KUKA KRL program: EPS_2_25089_SANMH02A_C_20251118074756.src

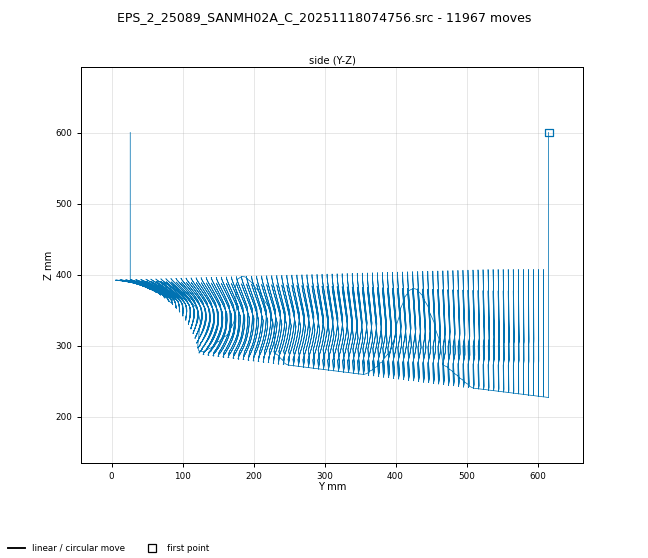
[picture p0: tool path of EPS_2_25089_SANMH02A_C_20251118074756.src, 11967 of 11969 moves have a stored position in this frame; points joined in program order, loops and branches not executed]
&ACCESS RVP
&REL 4
&COMMENT QRS 19112012
&PARAM EDITMASK = *
DEF PART()
EXT BAS (BAS_COMMAND :IN,REAL :IN )
INT I
BAS (#INITMOV,0 )

;KUKA QRS Post kuka4.cps  Date:22-06-2017 !

File_ID=2924

QRS_PRE_INIT()

;Init var - Until changes are made in qrs_pre_init
Outlet_Square_prg=0
Inlet_1_Square_prg=0
Inlet_2_Square_prg=0
Inlet_3_Square_prg=0
Inlet_4_Square_prg=0
Inlet_5_Square_prg=0

Outlet_1={X 0.000, Y 531.880, Z 306.500, B 0.000, E1 0.000 }
Inlet_1={X 0.000, Y 534.050, Z 276.500, B 0.000, E1 180.000 }
Outlet_1_type=201
Inlet_1_type=201
;QRS#1=Sidecore dimensions
;QRS#2=200-8" PVC SDR 35
;QRS#3=200-8" PVC SDR 35
;QRS#4=
;QRS#5=
;QRS#6=
;QRS#7=
;QRS#8=
;QRS#9=12-08 PSX
;QRS#10=12-08 PSX
;QRS#11=
;QRS#12=
;QRS#13=
;QRS#14=
;QRS#15=
;QRS#16=1220x127x686 2,25'
;QRS#17=EPS Height
;QRS#18=407
;QRS#19=*
;QRS#20= UPDATED VERSION 22-06-2017
;QRS#21=*
Outlet_Square=0100
Inlet_1_Square=0100
Inlet_2_Square=0
Inlet_3_Square=0
Inlet_4_Square=0
Inlet_5_Square=0
Mill_Square=1
Outlet_Square_Prg=204
Inlet_1_Square_prg=204

QRS_INIT()

$ADVANCE=5

; T1
PTP {E1 173.625,E2 173.625}
PTP {X 0,Y 615.476,A -85,B 0,C 180,E1 173.625,E2 173.625,E3 0,E4 0,E5 0,E6 0}
QRS_SPEED_INIT()
LIN {X 0,Y 615.476,Z 600,A -85,B 0,C 180,E1 173.625,E2 173.625,E3 0,E4 0,E5 0,E6 0} C_VEL
LIN {X 0,Y 615.476,Z 236.873,A -85,B 0,C 180,E1 173.625,E2 173.625} C_VEL
LIN {X 0,Y 615.476,Z 228.699,A -85,B 0,C 180,E1 173.625,E2 173.625} C_VEL
LIN {X 0,Y 615.468,Z 226.699,A -85,B 0,C 180,E1 173.439,E2 173.439} C_VEL
LIN {X 0,Y 615.497,Z 226.686,A -85,B 0,C 180,E1 170.801,E2 170.801} C_VEL
LIN {X 0,Y 615.491,Z 226.698,A -85,B 0,C 180,E1 168.139,E2 168.139} C_VEL
LIN {X 0,Y 615.457,Z 226.694,A -85,B 0,C 180,E1 165.45,E2 165.45} C_VEL
LIN {X 0,Y 615.478,Z 226.7,A -85,B 0,C 180,E1 162.729,E2 162.729} C_VEL
LIN {X 0,Y 615.448,Z 226.699,A -85,B 0,C 180,E1 159.966,E2 159.966} C_VEL
LIN {X 0,Y 615.489,Z 226.689,A -85,B 0,C 180,E1 157.155,E2 157.155} C_VEL
LIN {X 0,Y 615.498,Z 226.7,A -85,B 0,C 180,E1 154.285,E2 154.285} C_VEL
LIN {X 0,Y 615.471,Z 226.692,A -85,B 0,C 180,E1 151.553,E2 151.553} C_VEL
LIN {X 0,Y 615.467,Z 226.7,A -85,B 0,C 180,E1 148.917,E2 148.917} C_VEL
LIN {X 0,Y 615.436,Z 226.699,A -85,B 0,C 180,E1 146.473,E2 146.473} C_VEL
LIN {X 0,Y 615.483,Z 226.699,A -85,B 0,C 180,E1 144.167,E2 144.167} C_VEL
LIN {X 0,Y 615.486,Z 226.693,A -85,B 0,C 180,E1 141.931,E2 141.931} C_VEL
LIN {X 0,Y 615.489,Z 226.689,A -85,B 0,C 180,E1 139.393,E2 139.393} C_VEL
LIN {X 0,Y 615.461,Z 226.698,A -85,B 0,C 180,E1 136.753,E2 136.753} C_VEL
LIN {X 0,Y 615.469,Z 226.699,A -85,B 0,C 180,E1 133.995,E2 133.995} C_VEL
LIN {X 0,Y 615.461,Z 226.695,A -85,B 0,C 180,E1 131.476,E2 131.476} C_VEL
LIN {X 0,Y 615.472,Z 226.697,A -85,B 0,C 180,E1 128.906,E2 128.906} C_VEL
LIN {X 0,Y 615.482,Z 226.692,A -85,B 0,C 180,E1 126.425,E2 126.425} C_VEL
LIN {X 0,Y 615.484,Z 226.692,A -85,B 0,C 180,E1 125.616,E2 125.616} C_VEL
LIN {X 0,Y 615.472,Z 227.829,A -85,B 0,C 180,E1 124.698,E2 124.698} C_VEL
LIN {X 0,Y 615.474,Z 231.974,A -85,B 0,C 180,E1 122.328,E2 122.328} C_VEL
LIN {X 0,Y 615.461,Z 237.161,A -85,B 0,C 180,E1 119.408,E2 119.408} C_VEL
LIN {X 0,Y 615.486,Z 241.523,A -85,B 0,C 180,E1 117.044,E2 117.044} C_VEL
LIN {X 0,Y 615.488,Z 246.765,A -85,B 0,C 180,E1 114.272,E2 114.272} C_VEL
LIN {X 0,Y 615.472,Z 252.274,A -85,B 0,C 180,E1 111.432,E2 111.432} C_VEL
LIN {X 0,Y 615.494,Z 257.833,A -85,B 0,C 180,E1 108.605,E2 108.605} C_VEL
LIN {X 0,Y 615.465,Z 263.26,A -85,B 0,C 180,E1 105.906,E2 105.906} C_VEL
LIN {X 0,Y 615.491,Z 268.737,A -85,B 0,C 180,E1 103.201,E2 103.201} C_VEL
LIN {X 0,Y 615.483,Z 272.089,A -85,B 0,C 180,E1 101.569,E2 101.569} C_VEL
LIN {X 0,Y 615.49,Z 286.74,A -85,B 0,C 180,E1 101.235,E2 101.235} C_VEL
LIN {X 0,Y 615.492,Z 298.594,A -85,B 0,C 180,E1 100.843,E2 100.843} C_VEL
LIN {X 0,Y 615.473,Z 309.569,A -85,B 0,C 180,E1 100.361,E2 100.361} C_VEL
LIN {X 0,Y 615.483,Z 321.306,A -85,B 0,C 180,E1 99.696,E2 99.696} C_VEL
LIN {X 0,Y 615.499,Z 331.768,A -85,B 0,C 180,E1 98.95,E2 98.95} C_VEL
LIN {X 0,Y 615.498,Z 340.331,A -85,B 0,C 180,E1 98.206,E2 98.206} C_VEL
LIN {X 0,Y 615.497,Z 348.209,A -85,B 0,C 180,E1 97.38,E2 97.38} C_VEL
LIN {X 0,Y 615.497,Z 355.899,A -85,B 0,C 180,E1 96.392,E2 96.392} C_VEL
LIN {X 0,Y 615.497,Z 362.958,A -85,B 0,C 180,E1 95.241,E2 95.241} C_VEL
LIN {X 0,Y 615.493,Z 367.658,A -85,B 0,C 180,E1 94.256,E2 94.256} C_VEL
LIN {X 0,Y 615.495,Z 371.255,A -85,B 0,C 180,E1 93.273,E2 93.273} C_VEL
LIN {X 0,Y 615.496,Z 373.115,A -85,B 0,C 180,E1 92.618,E2 92.618} C_VEL
LIN {X 0,Y 615.497,Z 374.534,A -85,B 0,C 180,E1 91.963,E2 91.963} C_VEL
LIN {X 0,Y 615.496,Z 376.142,A -85,B 0,C 180,E1 90.654,E2 90.654} C_VEL
LIN {X 0,Y 615.494,Z 376.384,A -85,B 0,C 180,E1 90,E2 90} C_VEL
LIN {X 0,Y 615.495,Z 376.205,A -85,B 0,C 180,E1 89.346,E2 89.346} C_VEL
LIN {X 0,Y 615.496,Z 374.683,A -85,B 0,C 180,E1 88.037,E2 88.037} C_VEL
LIN {X 0,Y 615.498,Z 373.341,A -85,B 0,C 180,E1 87.382,E2 87.382} C_VEL
LIN {X 0,Y 615.496,Z 370.494,A -85,B 0,C 180,E1 86.399,E2 86.399} C_VEL
LIN {X 0,Y 615.498,Z 366.634,A -85,B 0,C 180,E1 85.415,E2 85.415} C_VEL
LIN {X 0,Y 615.498,Z 361.651,A -85,B 0,C 180,E1 84.43,E2 84.43} C_VEL
LIN {X 0,Y 615.497,Z 355.205,A -85,B 0,C 180,E1 83.417,E2 83.417} C_VEL
LIN {X 0,Y 615.497,Z 347.536,A -85,B 0,C 180,E1 82.455,E2 82.455} C_VEL
LIN {X 0,Y 615.498,Z 337.758,A -85,B 0,C 180,E1 81.463,E2 81.463} C_VEL
LIN {X 0,Y 615.498,Z 327.491,A -85,B 0,C 180,E1 80.636,E2 80.636} C_VEL
LIN {X 0,Y 615.469,Z 315.932,A -85,B 0,C 180,E1 79.888,E2 79.888} C_VEL
LIN {X 0,Y 615.492,Z 304.074,A -85,B 0,C 180,E1 79.293,E2 79.293} C_VEL
LIN {X 0,Y 615.485,Z 291.157,A -85,B 0,C 180,E1 78.807,E2 78.807} C_VEL
LIN {X 0,Y 615.486,Z 278.554,A -85,B 0,C 180,E1 78.473,E2 78.473} C_VEL
LIN {X 0,Y 615.486,Z 272.102,A -85,B 0,C 180,E1 78.348,E2 78.348} C_VEL
LIN {X 0,Y 615.487,Z 266.175,A -85,B 0,C 180,E1 75.451,E2 75.451} C_VEL
LIN {X 0,Y 615.496,Z 260.682,A -85,B 0,C 180,E1 72.73,E2 72.73} C_VEL
LIN {X 0,Y 615.469,Z 255.193,A -85,B 0,C 180,E1 69.966,E2 69.966} C_VEL
LIN {X 0,Y 615.487,Z 249.687,A -85,B 0,C 180,E1 67.155,E2 67.155} C_VEL
LIN {X 0,Y 615.466,Z 244.49,A -85,B 0,C 180,E1 64.436,E2 64.436} C_VEL
LIN {X 0,Y 615.474,Z 240.064,A -85,B 0,C 180,E1 62.084,E2 62.084} C_VEL
LIN {X 0,Y 615.5,Z 235.963,A -85,B 0,C 180,E1 59.84,E2 59.84} C_VEL
LIN {X 0,Y 615.46,Z 231.911,A -85,B 0,C 180,E1 57.541,E2 57.541} C_VEL
LIN {X 0,Y 615.469,Z 227.782,A -85,B 0,C 180,E1 55.183,E2 55.183} C_VEL
LIN {X 0,Y 615.487,Z 226.693,A -85,B 0,C 180,E1 54.384,E2 54.384} C_VEL
LIN {X 0,Y 615.488,Z 226.689,A -85,B 0,C 180,E1 51.931,E2 51.931} C_VEL
LIN {X 0,Y 615.476,Z 226.699,A -85,B 0,C 180,E1 49.392,E2 49.392} C_VEL
LIN {X 0,Y 615.436,Z 226.699,A -85,B 0,C 180,E1 46.958,E2 46.958} C_VEL
LIN {X 0,Y 615.485,Z 226.694,A -85,B 0,C 180,E1 44.15,E2 44.15} C_VEL
LIN {X 0,Y 615.466,Z 226.696,A -85,B 0,C 180,E1 41.476,E2 41.476} C_VEL
LIN {X 0,Y 615.481,Z 226.693,A -85,B 0,C 180,E1 38.905,E2 38.905} C_VEL
LIN {X 0,Y 615.487,Z 226.69,A -85,B 0,C 180,E1 36.425,E2 36.425} C_VEL
LIN {X 0,Y 615.478,Z 226.7,A -85,B 0,C 180,E1 34.023,E2 34.023} C_VEL
LIN {X 0,Y 615.432,Z 226.7,A -85,B 0,C 180,E1 31.689,E2 31.689} C_VEL
LIN {X 0,Y 615.459,Z 226.699,A -85,B 0,C 180,E1 29.408,E2 29.408} C_VEL
LIN {X 0,Y 615.477,Z 226.69,A -85,B 0,C 180,E1 26.445,E2 26.445} C_VEL
LIN {X 0,Y 615.488,Z 226.7,A -85,B 0,C 180,E1 24.008,E2 24.008} C_VEL
LIN {X 0,Y 615.463,Z 226.693,A -85,B 0,C 180,E1 21.433,E2 21.433} C_VEL
LIN {X 0,Y 615.472,Z 226.701,A -85,B 0,C 180,E1 18.6,E2 18.6} C_VEL
LIN {X 0,Y 615.443,Z 226.699,A -85,B 0,C 180,E1 15.906,E2 15.906} C_VEL
LIN {X 0,Y 615.494,Z 226.689,A -85,B 0,C 180,E1 13.201,E2 13.201} C_VEL
LIN {X 0,Y 615.481,Z 226.695,A -85,B 0,C 180,E1 10.527,E2 10.527} C_VEL
LIN {X 0,Y 615.466,Z 226.693,A -85,B 0,C 180,E1 7.876,E2 7.876} C_VEL
LIN {X 0,Y 615.496,Z 226.696,A -85,B 0,C 180,E1 5.241,E2 5.241} C_VEL
LIN {X 0,Y 615.433,Z 226.7,A -85,B 0,C 180,E1 2.618,E2 2.618} C_VEL
LIN {X 0,Y 615.484,Z 226.702,A -85,B 0,C 180,E1 0,E2 0} C_VEL
LIN {X 0,Y 615.485,Z 226.688,A -85,B 0,C 180,E1 -2.618,E2 -2.618} C_VEL
LIN {X 0,Y 615.49,Z 226.701,A -85,B 0,C 180,E1 -5.241,E2 -5.241} C_VEL
LIN {X 0,Y 615.462,Z 226.693,A -85,B 0,C 180,E1 -7.876,E2 -7.876} C_VEL
LIN {X 0,Y 615.441,Z 226.7,A -85,B 0,C 180,E1 -10.864,E2 -10.864} C_VEL
LIN {X 0,Y 615.447,Z 226.699,A -85,B 0,C 180,E1 -13.202,E2 -13.202} C_VEL
LIN {X 0,Y 615.494,Z 226.69,A -85,B 0,C 180,E1 -15.905,E2 -15.905} C_VEL
LIN {X 0,Y 615.486,Z 226.696,A -85,B 0,C 180,E1 -18.646,E2 -18.646} C_VEL
LIN {X 0,Y 615.465,Z 226.693,A -85,B 0,C 180,E1 -21.433,E2 -21.433} C_VEL
LIN {X 0,Y 615.467,Z 226.7,A -85,B 0,C 180,E1 -24.273,E2 -24.273} C_VEL
LIN {X 0,Y 615.438,Z 226.699,A -85,B 0,C 180,E1 -26.446,E2 -26.446} C_VEL
LIN {X 0,Y 615.457,Z 226.697,A -85,B 0,C 180,E1 -28.66,E2 -28.66} C_VEL
LIN {X 0,Y 615.487,Z 226.696,A -85,B 0,C 180,E1 -31.085,E2 -31.085} C_VEL
LIN {X 0,Y 615.488,Z 226.694,A -85,B 0,C 180,E1 -34.022,E2 -34.022} C_VEL
LIN {X 0,Y 615.46,Z 226.698,A -85,B 0,C 180,E1 -36.427,E2 -36.427} C_VEL
LIN {X 0,Y 615.457,Z 226.699,A -85,B 0,C 180,E1 -39.058,E2 -39.058} C_VEL
LIN {X 0,Y 615.485,Z 226.694,A -85,B 0,C 180,E1 -41.474,E2 -41.474} C_VEL
LIN {X 0,Y 615.467,Z 226.696,A -85,B 0,C 180,E1 -44.152,E2 -44.152} C_VEL
LIN {X 0,Y 615.483,Z 226.689,A -85,B 0,C 180,E1 -46.953,E2 -46.953} C_VEL
LIN {X 0,Y 615.478,Z 226.699,A -85,B 0,C 180,E1 -49.912,E2 -49.912} C_VEL
LIN {X 0,Y 615.445,Z 226.699,A -85,B 0,C 180,E1 -51.993,E2 -51.993} C_VEL
LIN {X 0,Y 615.465,Z 226.774,A -85,B 0,C 180,E1 -54.583,E2 -54.583} C_VEL
LIN {X 0,Y 615.487,Z 233.96,A -85,B 0,C 180,E1 -57.154,E2 -57.154} C_VEL
LIN {X 0,Y 615.452,Z 241.777,A -85,B 0,C 180,E1 -59.838,E2 -59.838} C_VEL
LIN {X 0,Y 615.493,Z 249.542,A -85,B 0,C 180,E1 -62.455,E2 -62.455} C_VEL
LIN {X 0,Y 615.47,Z 257.308,A -85,B 0,C 180,E1 -65.007,E2 -65.007} C_VEL
LIN {X 0,Y 615.475,Z 265.53,A -85,B 0,C 180,E1 -67.657,E2 -67.657} C_VEL
LIN {X 0,Y 615.486,Z 273.926,A -85,B 0,C 180,E1 -70.315,E2 -70.315} C_VEL
LIN {X 0,Y 615.488,Z 282.783,A -85,B 0,C 180,E1 -73.072,E2 -73.072} C_VEL
LIN {X 0,Y 615.46,Z 291.557,A -85,B 0,C 180,E1 -75.762,E2 -75.762} C_VEL
LIN {X 0,Y 615.498,Z 300.137,A -85,B 0,C 180,E1 -78.369,E2 -78.369} C_VEL
LIN {X 0,Y 615.497,Z 313.817,A -85,B 0,C 180,E1 -78.64,E2 -78.64} C_VEL
LIN {X 0,Y 615.451,Z 326.996,A -85,B 0,C 180,E1 -79.052,E2 -79.052} C_VEL
LIN {X 0,Y 615.438,Z 338.772,A -85,B 0,C 180,E1 -79.555,E2 -79.555} C_VEL
LIN {X 0,Y 615.482,Z 349.387,A -85,B 0,C 180,E1 -80.138,E2 -80.138} C_VEL
LIN {X 0,Y 615.498,Z 360.23,A -85,B 0,C 180,E1 -80.884,E2 -80.884} C_VEL
LIN {X 0,Y 615.497,Z 370.811,A -85,B 0,C 180,E1 -81.794,E2 -81.794} C_VEL
LIN {X 0,Y 615.498,Z 378.605,A -85,B 0,C 180,E1 -82.619,E2 -82.619} C_VEL
LIN {X 0,Y 615.496,Z 386.202,A -85,B 0,C 180,E1 -83.608,E2 -83.608} C_VEL
LIN {X 0,Y 615.498,Z 393.204,A -85,B 0,C 180,E1 -84.759,E2 -84.759} C_VEL
LIN {X 0,Y 615.494,Z 397.851,A -85,B 0,C 180,E1 -85.744,E2 -85.744} C_VEL
LIN {X 0,Y 615.494,Z 401.398,A -85,B 0,C 180,E1 -86.727,E2 -86.727} C_VEL
LIN {X 0,Y 615.497,Z 403.233,A -85,B 0,C 180,E1 -87.382,E2 -87.382} C_VEL
LIN {X 0,Y 615.5,Z 404.607,A -85,B 0,C 180,E1 -88.037,E2 -88.037} C_VEL
LIN {X 0,Y 615.496,Z 406.173,A -85,B 0,C 180,E1 -89.346,E2 -89.346} C_VEL
LIN {X 0,Y 615.494,Z 406.389,A -85,B 0,C 180,E1 -90,E2 -90} C_VEL
LIN {X 0,Y 615.495,Z 405.58,A -85,B 0,C 180,E1 -91.309,E2 -91.309} C_VEL
LIN {X 0,Y 615.5,Z 404.608,A -85,B 0,C 180,E1 -91.963,E2 -91.963} C_VEL
LIN {X 0,Y 615.497,Z 403.233,A -85,B 0,C 180,E1 -92.618,E2 -92.618} C_VEL
LIN {X 0,Y 615.496,Z 400.35,A -85,B 0,C 180,E1 -93.601,E2 -93.601} C_VEL
LIN {X 0,Y 615.498,Z 396.442,A -85,B 0,C 180,E1 -94.584,E2 -94.584} C_VEL
LIN {X 0,Y 615.499,Z 391.405,A -85,B 0,C 180,E1 -95.57,E2 -95.57} C_VEL
LIN {X 0,Y 615.497,Z 384.869,A -85,B 0,C 180,E1 -96.583,E2 -96.583} C_VEL
LIN {X 0,Y 615.497,Z 377.133,A -85,B 0,C 180,E1 -97.545,E2 -97.545} C_VEL
LIN {X 0,Y 615.498,Z 369.045,A -85,B 0,C 180,E1 -98.371,E2 -98.371} C_VEL
LIN {X 0,Y 615.499,Z 359.168,A -85,B 0,C 180,E1 -99.199,E2 -99.199} C_VEL
LIN {X 0,Y 615.472,Z 347.985,A -85,B 0,C 180,E1 -99.945,E2 -99.945} C_VEL
LIN {X 0,Y 615.437,Z 337.031,A -85,B 0,C 180,E1 -100.528,E2 -100.528} C_VEL
LIN {X 0,Y 615.457,Z 324.794,A -85,B 0,C 180,E1 -101.03,E2 -101.03} C_VEL
LIN {X 0,Y 615.499,Z 312.064,A -85,B 0,C 180,E1 -101.401,E2 -101.401} C_VEL
LIN {X 0,Y 615.498,Z 300.137,A -85,B 0,C 180,E1 -101.631,E2 -101.631} C_VEL
LIN {X 0,Y 615.46,Z 291.557,A -85,B 0,C 180,E1 -104.238,E2 -104.238} C_VEL
LIN {X 0,Y 615.488,Z 282.784,A -85,B 0,C 180,E1 -106.928,E2 -106.928} C_VEL
LIN {X 0,Y 615.486,Z 273.927,A -85,B 0,C 180,E1 -109.685,E2 -109.685} C_VEL
LIN {X 0,Y 615.479,Z 265.527,A -85,B 0,C 180,E1 -112.343,E2 -112.343} C_VEL
LIN {X 0,Y 615.47,Z 257.308,A -85,B 0,C 180,E1 -114.993,E2 -114.993} C_VEL
LIN {X 0,Y 615.453,Z 248.44,A -85,B 0,C 180,E1 -117.917,E2 -117.917} C_VEL
LIN {X 0,Y 615.473,Z 240.656,A -85,B 0,C 180,E1 -120.54,E2 -120.54} C_VEL
LIN {X 0,Y 615.491,Z 232.848,A -85,B 0,C 180,E1 -123.236,E2 -123.236} C_VEL
LIN {X 0,Y 615.46,Z 226.7,A -85,B 0,C 180,E1 -125.467,E2 -125.467} C_VEL
LIN {X 0,Y 615.448,Z 226.699,A -85,B 0,C 180,E1 -128.072,E2 -128.072} C_VEL
LIN {X 0,Y 615.491,Z 226.693,A -85,B 0,C 180,E1 -130.606,E2 -130.606} C_VEL
LIN {X 0,Y 615.479,Z 226.692,A -85,B 0,C 180,E1 -133.245,E2 -133.245} C_VEL
LIN {X 0,Y 615.463,Z 226.695,A -85,B 0,C 180,E1 -136.005,E2 -136.005} C_VEL
LIN {X 0,Y 615.483,Z 226.702,A -85,B 0,C 180,E1 -138.906,E2 -138.906} C_VEL
LIN {X 0,Y 615.455,Z 226.7,A -85,B 0,C 180,E1 -141.929,E2 -141.929} C_VEL
LIN {X 0,Y 615.496,Z 226.69,A -85,B 0,C 180,E1 -144.385,E2 -144.385} C_VEL
LIN {X 0,Y 615.479,Z 226.69,A -85,B 0,C 180,E1 -146.763,E2 -146.763} C_VEL
LIN {X 0,Y 615.496,Z 226.699,A -85,B 0,C 180,E1 -149.081,E2 -149.081} C_VEL
LIN {X 0,Y 615.454,Z 226.696,A -85,B 0,C 180,E1 -151.556,E2 -151.556} C_VEL
LIN {X 0,Y 615.477,Z 226.7,A -85,B 0,C 180,E1 -154.434,E2 -154.434} C_VEL
LIN {X 0,Y 615.448,Z 226.698,A -85,B 0,C 180,E1 -157.154,E2 -157.154} C_VEL
LIN {X 0,Y 615.489,Z 226.689,A -85,B 0,C 180,E1 -159.967,E2 -159.967} C_VEL
LIN {X 0,Y 615.489,Z 226.698,A -85,B 0,C 180,E1 -162.729,E2 -162.729} C_VEL
LIN {X 0,Y 615.464,Z 226.693,A -85,B 0,C 180,E1 -165.45,E2 -165.45} C_VEL
LIN {X 0,Y 615.48,Z 226.7,A -85,B 0,C 180,E1 -168.139,E2 -168.139} C_VEL
LIN {X 0,Y 615.441,Z 226.699,A -85,B 0,C 180,E1 -170.801,E2 -170.801} C_VEL
LIN {X 0,Y 615.493,Z 226.693,A -85,B 0,C 180,E1 -173.443,E2 -173.443} C_VEL
LIN {X 0,Y 615.479,Z 226.692,A -85,B 0,C 180,E1 -176.071,E2 -176.071} C_VEL
LIN {X 0,Y 615.467,Z 226.696,A -85,B 0,C 180,E1 -178.691,E2 -178.691} C_VEL
LIN {X 0,Y 615.482,Z 226.693,A -85,B 0,C 180,E1 -181.309,E2 -181.309} C_VEL
LIN {X 0,Y 615.443,Z 226.7,A -85,B 0,C 180,E1 -183.929,E2 -183.929} C_VEL
LIN {X 0,Y 615.452,Z 226.696,A -85,B 0,C 180,E1 -185.899,E2 -185.899} C_VEL
LIN {X 0,Y 615.468,Z 226.699,A -85,B 0,C 180,E1 -186.561,E2 -186.561} C_VEL
LIN {X 0,Y 614.809,Z 226.842,A -85,B 0,C 180,E1 -187.107,E2 -187.107} C_VEL
LIN {X 0,Y 611.991,Z 227.25,A -85,B 0,C 180,E1 -187.993,E2 -187.993} C_VEL
LIN {X 0,Y 609.601,Z 227.559,A -85,B 0,C 180,E1 -188.705,E2 -188.705} C_VEL
LIN {X 0,Y 608.558,Z 227.678,A -85,B 0,C 180,E1 -189.255,E2 -189.255} C_VEL
LIN {X 0,Y 608.465,Z 227.689,A -85,B 0,C 180,E1 -189.441,E2 -189.441} C_VEL
LIN {X 0,Y 608.463,Z 227.697,A -85,B 0,C 180,E1 -192,E2 -192} C_VEL
LIN {X 0,Y 608.431,Z 227.693,A -85,B 0,C 180,E1 -194.722,E2 -194.722} C_VEL
LIN {X 0,Y 608.431,Z 227.696,A -85,B 0,C 180,E1 -197.477,E2 -197.477} C_VEL
LIN {X 0,Y 608.424,Z 227.694,A -85,B 0,C 180,E1 -199.572,E2 -199.572} C_VEL
LIN {X 0,Y 608.453,Z 227.691,A -85,B 0,C 180,E1 -201.692,E2 -201.692} C_VEL
LIN {X 0,Y 608.454,Z 227.691,A -85,B 0,C 180,E1 -204.571,E2 -204.571} C_VEL
LIN {X 0,Y 608.482,Z 227.691,A -85,B 0,C 180,E1 -207.208,E2 -207.208} C_VEL
LIN {X 0,Y 608.414,Z 227.695,A -85,B 0,C 180,E1 -209.963,E2 -209.963} C_VEL
LIN {X 0,Y 608.457,Z 227.697,A -85,B 0,C 180,E1 -212.521,E2 -212.521} C_VEL
LIN {X 0,Y 608.426,Z 227.694,A -85,B 0,C 180,E1 -215.279,E2 -215.279} C_VEL
LIN {X 0,Y 608.467,Z 227.689,A -85,B 0,C 180,E1 -218.24,E2 -218.24} C_VEL
LIN {X 0,Y 608.455,Z 227.694,A -85,B 0,C 180,E1 -221.341,E2 -221.341} C_VEL
LIN {X 0,Y 608.452,Z 227.694,A -85,B 0,C 180,E1 -224.263,E2 -224.263} C_VEL
LIN {X 0,Y 608.404,Z 227.696,A -85,B 0,C 180,E1 -227.036,E2 -227.036} C_VEL
LIN {X 0,Y 608.455,Z 227.698,A -85,B 0,C 180,E1 -229.697,E2 -229.697} C_VEL
LIN {X 0,Y 608.467,Z 227.688,A -85,B 0,C 180,E1 -232.254,E2 -232.254} C_VEL
LIN {X 0,Y 608.41,Z 227.816,A -85,B 0,C 180,E1 -234.72,E2 -234.72} C_VEL
LIN {X 0,Y 608.439,Z 231.95,A -85,B 0,C 180,E1 -237.119,E2 -237.119} C_VEL
LIN {X 0,Y 608.444,Z 237.072,A -85,B 0,C 180,E1 -240.033,E2 -240.033} C_VEL
LIN {X 0,Y 608.426,Z 242.105,A -85,B 0,C 180,E1 -242.803,E2 -242.803} C_VEL
LIN {X 0,Y 608.427,Z 247.036,A -85,B 0,C 180,E1 -245.428,E2 -245.428} C_VEL
LIN {X 0,Y 608.436,Z 251.183,A -85,B 0,C 180,E1 -247.593,E2 -247.593} C_VEL
LIN {X 0,Y 608.426,Z 256.713,A -85,B 0,C 180,E1 -250.429,E2 -250.429} C_VEL
LIN {X 0,Y 608.45,Z 262.242,A -85,B 0,C 180,E1 -253.216,E2 -253.216} C_VEL
LIN {X 0,Y 608.418,Z 267.858,A -85,B 0,C 180,E1 -256.004,E2 -256.004} C_VEL
LIN {X 0,Y 608.434,Z 272.524,A -85,B 0,C 180,E1 -258.296,E2 -258.296} C_VEL
LIN {X 0,Y 608.53,Z 288.393,A -85,B 0,C 180,E1 -258.677,E2 -258.677} C_VEL
LIN {X 0,Y 608.534,Z 300.772,A -85,B 0,C 180,E1 -259.112,E2 -259.112} C_VEL
LIN {X 0,Y 608.473,Z 312.935,A -85,B 0,C 180,E1 -259.687,E2 -259.687} C_VEL
LIN {X 0,Y 608.49,Z 324.067,A -85,B 0,C 180,E1 -260.359,E2 -260.359} C_VEL
LIN {X 0,Y 608.474,Z 333.084,A -85,B 0,C 180,E1 -261.029,E2 -261.029} C_VEL
LIN {X 0,Y 608.464,Z 342.35,A -85,B 0,C 180,E1 -261.866,E2 -261.866} C_VEL
LIN {X 0,Y 608.466,Z 351.324,A -85,B 0,C 180,E1 -262.867,E2 -262.867} C_VEL
LIN {X 0,Y 608.444,Z 358.556,A -85,B 0,C 180,E1 -263.867,E2 -263.867} C_VEL
LIN {X 0,Y 608.462,Z 363.435,A -85,B 0,C 180,E1 -264.698,E2 -264.698} C_VEL
LIN {X 0,Y 608.439,Z 368.178,A -85,B 0,C 180,E1 -265.694,E2 -265.694} C_VEL
LIN {X 0,Y 608.425,Z 371.812,A -85,B 0,C 180,E1 -266.689,E2 -266.689} C_VEL
LIN {X 0,Y 608.425,Z 373.691,A -85,B 0,C 180,E1 -267.352,E2 -267.352} C_VEL
LIN {X 0,Y 608.442,Z 375.127,A -85,B 0,C 180,E1 -268.014,E2 -268.014} C_VEL
LIN {X 0,Y 608.439,Z 376.752,A -85,B 0,C 180,E1 -269.338,E2 -269.338} C_VEL
LIN {X 0,Y 608.434,Z 376.995,A -85,B 0,C 180,E1 -270,E2 -270} C_VEL
LIN {X 0,Y 608.438,Z 376.815,A -85,B 0,C 180,E1 -270.662,E2 -270.662} C_VEL
LIN {X 0,Y 608.441,Z 375.276,A -85,B 0,C 180,E1 -271.986,E2 -271.986} C_VEL
LIN {X 0,Y 608.427,Z 373.918,A -85,B 0,C 180,E1 -272.648,E2 -272.648} C_VEL
LIN {X 0,Y 608.449,Z 371.041,A -85,B 0,C 180,E1 -273.642,E2 -273.642} C_VEL
LIN {X 0,Y 608.433,Z 367.142,A -85,B 0,C 180,E1 -274.638,E2 -274.638} C_VEL
LIN {X 0,Y 608.449,Z 362.112,A -85,B 0,C 180,E1 -275.635,E2 -275.635} C_VEL
LIN {X 0,Y 608.442,Z 355.794,A -85,B 0,C 180,E1 -276.633,E2 -276.633} C_VEL
LIN {X 0,Y 608.475,Z 347.878,A -85,B 0,C 180,E1 -277.633,E2 -277.633} C_VEL
LIN {X 0,Y 608.472,Z 338.035,A -85,B 0,C 180,E1 -278.636,E2 -278.636} C_VEL
LIN {X 0,Y 608.481,Z 327.712,A -85,B 0,C 180,E1 -279.473,E2 -279.473} C_VEL
LIN {X 0,Y 608.466,Z 316.098,A -85,B 0,C 180,E1 -280.229,E2 -280.229} C_VEL
LIN {X 0,Y 608.508,Z 304.205,A -85,B 0,C 180,E1 -280.831,E2 -280.831} C_VEL
LIN {X 0,Y 608.527,Z 291.258,A -85,B 0,C 180,E1 -281.323,E2 -281.323} C_VEL
LIN {X 0,Y 608.538,Z 278.64,A -85,B 0,C 180,E1 -281.66,E2 -281.66} C_VEL
LIN {X 0,Y 608.435,Z 272.535,A -85,B 0,C 180,E1 -281.789,E2 -281.789} C_VEL
LIN {X 0,Y 608.419,Z 266.571,A -85,B 0,C 180,E1 -284.722,E2 -284.722} C_VEL
LIN {X 0,Y 608.434,Z 261.039,A -85,B 0,C 180,E1 -287.477,E2 -287.477} C_VEL
LIN {X 0,Y 608.423,Z 255.506,A -85,B 0,C 180,E1 -290.276,E2 -290.276} C_VEL
LIN {X 0,Y 608.429,Z 249.974,A -85,B 0,C 180,E1 -293.125,E2 -293.125} C_VEL
LIN {X 0,Y 608.435,Z 244.44,A -85,B 0,C 180,E1 -296.036,E2 -296.036} C_VEL
LIN {X 0,Y 608.443,Z 239.653,A -85,B 0,C 180,E1 -298.614,E2 -298.614} C_VEL
LIN {X 0,Y 608.401,Z 234.851,A -85,B 0,C 180,E1 -301.32,E2 -301.32} C_VEL
LIN {X 0,Y 608.449,Z 230.643,A -85,B 0,C 180,E1 -303.731,E2 -303.731} C_VEL
LIN {X 0,Y 608.438,Z 227.967,A -85,B 0,C 180,E1 -305.278,E2 -305.278} C_VEL
LIN {X 0,Y 608.477,Z 227.692,A -85,B 0,C 180,E1 -307.159,E2 -307.159} C_VEL
LIN {X 0,Y 608.439,Z 227.692,A -85,B 0,C 180,E1 -309.442,E2 -309.442} C_VEL
LIN {X 0,Y 608.44,Z 227.696,A -85,B 0,C 180,E1 -312.332,E2 -312.332} C_VEL
LIN {X 0,Y 608.414,Z 227.695,A -85,B 0,C 180,E1 -314.8,E2 -314.8} C_VEL
LIN {X 0,Y 608.438,Z 227.697,A -85,B 0,C 180,E1 -317.039,E2 -317.039} C_VEL
LIN {X 0,Y 608.456,Z 227.69,A -85,B 0,C 180,E1 -319.697,E2 -319.697} C_VEL
LIN {X 0,Y 608.466,Z 227.695,A -85,B 0,C 180,E1 -322.253,E2 -322.253} C_VEL
LIN {X 0,Y 608.437,Z 227.692,A -85,B 0,C 180,E1 -325.097,E2 -325.097} C_VEL
LIN {X 0,Y 608.446,Z 227.693,A -85,B 0,C 180,E1 -327.904,E2 -327.904} C_VEL
LIN {X 0,Y 608.46,Z 227.697,A -85,B 0,C 180,E1 -330.98,E2 -330.98} C_VEL
LIN {X 0,Y 608.448,Z 227.692,A -85,B 0,C 180,E1 -333.226,E2 -333.226} C_VEL
LIN {X 0,Y 608.48,Z 227.691,A -85,B 0,C 180,E1 -335.848,E2 -335.848} C_VEL
LIN {X 0,Y 608.456,Z 227.691,A -85,B 0,C 180,E1 -338.308,E2 -338.308} C_VEL
LIN {X 0,Y 608.448,Z 227.697,A -85,B 0,C 180,E1 -341.13,E2 -341.13} C_VEL
LIN {X 0,Y 608.42,Z 227.694,A -85,B 0,C 180,E1 -343.905,E2 -343.905} C_VEL
LIN {X 0,Y 608.467,Z 227.692,A -85,B 0,C 180,E1 -346.644,E2 -346.644} C_VEL
LIN {X 0,Y 608.46,Z 227.691,A -85,B 0,C 180,E1 -349.35,E2 -349.35} C_VEL
LIN {X 0,Y 608.436,Z 227.693,A -85,B 0,C 180,E1 -352.032,E2 -352.032} C_VEL
LIN {X 0,Y 608.471,Z 227.692,A -85,B 0,C 180,E1 -354.698,E2 -354.698} C_VEL
LIN {X 0,Y 608.43,Z 227.693,A -85,B 0,C 180,E1 -357.352,E2 -357.352} C_VEL
LIN {X 0,Y 608.475,Z 227.695,A -85,B 0,C 180,E1 -360,E2 -360} C_VEL
LIN {X 0,Y 608.477,Z 227.687,A -85,B 0,C 180,E1 -362.648,E2 -362.648} C_VEL
LIN {X 0,Y 608.468,Z 227.695,A -85,B 0,C 180,E1 -365.302,E2 -365.302} C_VEL
LIN {X 0,Y 608.434,Z 227.693,A -85,B 0,C 180,E1 -367.968,E2 -367.968} C_VEL
LIN {X 0,Y 608.44,Z 227.695,A -85,B 0,C 180,E1 -370.65,E2 -370.65} C_VEL
LIN {X 0,Y 608.438,Z 227.694,A -85,B 0,C 180,E1 -373.357,E2 -373.357} C_VEL
LIN {X 0,Y 608.461,Z 227.69,A -85,B 0,C 180,E1 -376.094,E2 -376.094} C_VEL
LIN {X 0,Y 608.455,Z 227.698,A -85,B 0,C 180,E1 -378.87,E2 -378.87} C_VEL
LIN {X 0,Y 608.46,Z 227.69,A -85,B 0,C 180,E1 -381.692,E2 -381.692} C_VEL
LIN {X 0,Y 608.425,Z 227.695,A -85,B 0,C 180,E1 -384.572,E2 -384.572} C_VEL
LIN {X 0,Y 608.461,Z 227.693,A -85,B 0,C 180,E1 -387.203,E2 -387.203} C_VEL
LIN {X 0,Y 608.446,Z 227.691,A -85,B 0,C 180,E1 -389.967,E2 -389.967} C_VEL
LIN {X 0,Y 608.462,Z 227.696,A -85,B 0,C 180,E1 -392.522,E2 -392.522} C_VEL
LIN {X 0,Y 608.441,Z 227.692,A -85,B 0,C 180,E1 -395.278,E2 -395.278} C_VEL
LIN {X 0,Y 608.453,Z 227.698,A -85,B 0,C 180,E1 -397.748,E2 -397.748} C_VEL
LIN {X 0,Y 608.404,Z 227.696,A -85,B 0,C 180,E1 -400.323,E2 -400.323} C_VEL
LIN {X 0,Y 608.457,Z 227.696,A -85,B 0,C 180,E1 -402.96,E2 -402.96} C_VEL
LIN {X 0,Y 608.448,Z 227.692,A -85,B 0,C 180,E1 -405.737,E2 -405.737} C_VEL
LIN {X 0,Y 608.452,Z 227.691,A -85,B 0,C 180,E1 -408.659,E2 -408.659} C_VEL
LIN {X 0,Y 608.435,Z 227.7,A -85,B 0,C 180,E1 -411.409,E2 -411.409} C_VEL
LIN {X 0,Y 608.429,Z 227.694,A -85,B 0,C 180,E1 -413.957,E2 -413.957} C_VEL
LIN {X 0,Y 608.483,Z 227.878,A -85,B 0,C 180,E1 -414.522,E2 -414.522} C_VEL
LIN {X 0,Y 608.496,Z 235.07,A -85,B 0,C 180,E1 -417.123,E2 -417.123} C_VEL
LIN {X 0,Y 608.46,Z 243.499,A -85,B 0,C 180,E1 -420.03,E2 -420.03} C_VEL
LIN {X 0,Y 608.476,Z 251.679,A -85,B 0,C 180,E1 -422.794,E2 -422.794} C_VEL
LIN {X 0,Y 608.439,Z 259.656,A -85,B 0,C 180,E1 -425.428,E2 -425.428} C_VEL
LIN {X 0,Y 608.455,Z 267.447,A -85,B 0,C 180,E1 -427.951,E2 -427.951} C_VEL
LIN {X 0,Y 608.457,Z 276.352,A -85,B 0,C 180,E1 -430.78,E2 -430.78} C_VEL
LIN {X 0,Y 608.431,Z 285.008,A -85,B 0,C 180,E1 -433.484,E2 -433.484} C_VEL
LIN {X 0,Y 608.443,Z 294.216,A -85,B 0,C 180,E1 -436.32,E2 -436.32} C_VEL
LIN {X 0,Y 608.436,Z 300.491,A -85,B 0,C 180,E1 -438.232,E2 -438.232} C_VEL
LIN {X 0,Y 608.546,Z 314.693,A -85,B 0,C 180,E1 -438.53,E2 -438.53} C_VEL
LIN {X 0,Y 608.494,Z 327.82,A -85,B 0,C 180,E1 -438.951,E2 -438.951} C_VEL
LIN {X 0,Y 608.467,Z 338.919,A -85,B 0,C 180,E1 -439.434,E2 -439.434} C_VEL
LIN {X 0,Y 608.471,Z 349.577,A -85,B 0,C 180,E1 -440.023,E2 -440.023} C_VEL
LIN {X 0,Y 608.483,Z 360.473,A -85,B 0,C 180,E1 -440.778,E2 -440.778} C_VEL
LIN {X 0,Y 608.475,Z 371.111,A -85,B 0,C 180,E1 -441.699,E2 -441.699} C_VEL
LIN {X 0,Y 608.471,Z 378.959,A -85,B 0,C 180,E1 -442.534,E2 -442.534} C_VEL
LIN {X 0,Y 608.461,Z 386.286,A -85,B 0,C 180,E1 -443.484,E2 -443.484} C_VEL
LIN {X 0,Y 608.451,Z 391.865,A -85,B 0,C 180,E1 -444.366,E2 -444.366} C_VEL
LIN {X 0,Y 608.432,Z 396.95,A -85,B 0,C 180,E1 -445.362,E2 -445.362} C_VEL
LIN {X 0,Y 608.449,Z 400.896,A -85,B 0,C 180,E1 -446.358,E2 -446.358} C_VEL
LIN {X 0,Y 608.425,Z 403.809,A -85,B 0,C 180,E1 -447.352,E2 -447.352} C_VEL
LIN {X 0,Y 608.444,Z 405.201,A -85,B 0,C 180,E1 -448.014,E2 -448.014} C_VEL
LIN {X 0,Y 608.438,Z 406.783,A -85,B 0,C 180,E1 -449.338,E2 -449.338} C_VEL
LIN {X 0,Y 608.434,Z 407,A -85,B 0,C 180,E1 -450,E2 -450} C_VEL
LIN {X 0,Y 608.448,Z 406.184,A -85,B 0,C 180,E1 -451.324,E2 -451.324} C_VEL
LIN {X 0,Y 608.444,Z 405.201,A -85,B 0,C 180,E1 -451.986,E2 -451.986} C_VEL
LIN {X 0,Y 608.425,Z 403.809,A -85,B 0,C 180,E1 -452.648,E2 -452.648} C_VEL
LIN {X 0,Y 608.449,Z 400.896,A -85,B 0,C 180,E1 -453.642,E2 -453.642} C_VEL
LIN {X 0,Y 608.432,Z 396.95,A -85,B 0,C 180,E1 -454.638,E2 -454.638} C_VEL
LIN {X 0,Y 608.438,Z 390.877,A -85,B 0,C 180,E1 -455.801,E2 -455.801} C_VEL
LIN {X 0,Y 608.462,Z 384.235,A -85,B 0,C 180,E1 -456.799,E2 -456.799} C_VEL
LIN {X 0,Y 608.456,Z 375.989,A -85,B 0,C 180,E1 -457.8,E2 -457.8} C_VEL
LIN {X 0,Y 608.472,Z 367.537,A -85,B 0,C 180,E1 -458.636,E2 -458.636} C_VEL
LIN {X 0,Y 608.48,Z 357.091,A -85,B 0,C 180,E1 -459.473,E2 -459.473} C_VEL
LIN {X 0,Y 608.482,Z 346.756,A -85,B 0,C 180,E1 -460.145,E2 -460.145} C_VEL
LIN {X 0,Y 608.463,Z 335.872,A -85,B 0,C 180,E1 -460.712,E2 -460.712} C_VEL
LIN {X 0,Y 608.492,Z 324.1,A -85,B 0,C 180,E1 -461.186,E2 -461.186} C_VEL
LIN {X 0,Y 608.551,Z 311.267,A -85,B 0,C 180,E1 -461.554,E2 -461.554} C_VEL
LIN {X 0,Y 608.436,Z 300.492,A -85,B 0,C 180,E1 -461.768,E2 -461.768} C_VEL
LIN {X 0,Y 608.407,Z 291.935,A -85,B 0,C 180,E1 -464.38,E2 -464.38} C_VEL
LIN {X 0,Y 608.452,Z 284.144,A -85,B 0,C 180,E1 -466.784,E2 -466.784} C_VEL
LIN {X 0,Y 608.459,Z 275.239,A -85,B 0,C 180,E1 -469.57,E2 -469.57} C_VEL
LIN {X 0,Y 608.462,Z 266.116,A -85,B 0,C 180,E1 -472.476,E2 -472.476} C_VEL
LIN {X 0,Y 608.451,Z 257.43,A -85,B 0,C 180,E1 -475.301,E2 -475.301} C_VEL
LIN {X 0,Y 608.441,Z 249.639,A -85,B 0,C 180,E1 -477.892,E2 -477.892} C_VEL
LIN {X 0,Y 608.473,Z 241.817,A -85,B 0,C 180,E1 -480.545,E2 -480.545} C_VEL
LIN {X 0,Y 608.49,Z 233.958,A -85,B 0,C 180,E1 -483.272,E2 -483.272} C_VEL
LIN {X 0,Y 608.428,Z 227.697,A -85,B 0,C 180,E1 -485.583,E2 -485.583} C_VEL
LIN {X 0,Y 608.442,Z 227.695,A -85,B 0,C 180,E1 -488.237,E2 -488.237} C_VEL
LIN {X 0,Y 608.448,Z 227.691,A -85,B 0,C 180,E1 -491.177,E2 -491.177} C_VEL
LIN {X 0,Y 608.466,Z 227.694,A -85,B 0,C 180,E1 -493.87,E2 -493.87} C_VEL
LIN {X 0,Y 608.483,Z 227.688,A -85,B 0,C 180,E1 -496.69,E2 -496.69} C_VEL
LIN {X 0,Y 608.451,Z 227.698,A -85,B 0,C 180,E1 -498.823,E2 -498.823} C_VEL
LIN {X 0,Y 608.414,Z 227.696,A -85,B 0,C 180,E1 -501.766,E2 -501.766} C_VEL
LIN {X 0,Y 608.449,Z 227.698,A -85,B 0,C 180,E1 -503.954,E2 -503.954} C_VEL
LIN {X 0,Y 608.47,Z 227.689,A -85,B 0,C 180,E1 -506.33,E2 -506.33} C_VEL
LIN {X 0,Y 608.48,Z 227.689,A -85,B 0,C 180,E1 -508.728,E2 -508.728} C_VEL
LIN {X 0,Y 608.448,Z 227.692,A -85,B 0,C 180,E1 -511.385,E2 -511.385} C_VEL
LIN {X 0,Y 608.475,Z 227.695,A -85,B 0,C 180,E1 -514.279,E2 -514.279} C_VEL
LIN {X 0,Y 608.424,Z 227.694,A -85,B 0,C 180,E1 -516.875,E2 -516.875} C_VEL
LIN {X 0,Y 608.468,Z 227.695,A -85,B 0,C 180,E1 -519.322,E2 -519.322} C_VEL
LIN {X 0,Y 608.453,Z 227.69,A -85,B 0,C 180,E1 -521.828,E2 -521.828} C_VEL
LIN {X 0,Y 608.468,Z 227.696,A -85,B 0,C 180,E1 -524.594,E2 -524.594} C_VEL
LIN {X 0,Y 608.449,Z 227.691,A -85,B 0,C 180,E1 -527.322,E2 -527.322} C_VEL
LIN {X 0,Y 608.432,Z 227.696,A -85,B 0,C 180,E1 -530.022,E2 -530.022} C_VEL
LIN {X 0,Y 608.434,Z 227.694,A -85,B 0,C 180,E1 -532.7,E2 -532.7} C_VEL
LIN {X 0,Y 608.457,Z 227.691,A -85,B 0,C 180,E1 -535.362,E2 -535.362} C_VEL
LIN {X 0,Y 608.459,Z 227.693,A -85,B 0,C 180,E1 -538.014,E2 -538.014} C_VEL
LIN {X 0,Y 608.449,Z 227.691,A -85,B 0,C 180,E1 -540.662,E2 -540.662} C_VEL
LIN {X 0,Y 608.467,Z 227.695,A -85,B 0,C 180,E1 -543.311,E2 -543.311} C_VEL
LIN {X 0,Y 608.429,Z 227.693,A -85,B 0,C 180,E1 -545.967,E2 -545.967} C_VEL
LIN {X 0,Y 608.461,Z 227.696,A -85,B 0,C 180,E1 -548.636,E2 -548.636} C_VEL
LIN {X 0,Y 608.465,Z 227.689,A -85,B 0,C 180,E1 -549.441,E2 -549.441} C_VEL
LIN {X 0,Y 607.776,Z 227.779,A -85,B 0,C 180,E1 -549.994,E2 -549.994} C_VEL
LIN {X 0,Y 604.922,Z 228.136,A -85,B 0,C 180,E1 -550.891,E2 -550.891} C_VEL
LIN {X 0,Y 602.523,Z 228.436,A -85,B 0,C 180,E1 -551.612,E2 -551.612} C_VEL
LIN {X 0,Y 601.492,Z 228.563,A -85,B 0,C 180,E1 -552.169,E2 -552.169} C_VEL
LIN {X 0,Y 601.407,Z 228.571,A -85,B 0,C 180,E1 -552.357,E2 -552.357} C_VEL
LIN {X 0,Y 601.401,Z 228.57,A -85,B 0,C 180,E1 -554.898,E2 -554.898} C_VEL
LIN {X 0,Y 601.402,Z 228.574,A -85,B 0,C 180,E1 -556.987,E2 -556.987} C_VEL
LIN {X 0,Y 601.385,Z 228.571,A -85,B 0,C 180,E1 -559.81,E2 -559.81} C_VEL
LIN {X 0,Y 601.407,Z 228.571,A -85,B 0,C 180,E1 -561.96,E2 -561.96} C_VEL
LIN {X 0,Y 601.439,Z 228.567,A -85,B 0,C 180,E1 -564.293,E2 -564.293} C_VEL
LIN {X 0,Y 601.454,Z 228.566,A -85,B 0,C 180,E1 -567.111,E2 -567.111} C_VEL
LIN {X 0,Y 601.399,Z 228.573,A -85,B 0,C 180,E1 -569.394,E2 -569.394} C_VEL
LIN {X 0,Y 601.386,Z 228.57,A -85,B 0,C 180,E1 -571.728,E2 -571.728} C_VEL
LIN {X 0,Y 601.411,Z 228.573,A -85,B 0,C 180,E1 -574.12,E2 -574.12} C_VEL
LIN {X 0,Y 601.396,Z 228.57,A -85,B 0,C 180,E1 -576.584,E2 -576.584} C_VEL
LIN {X 0,Y 601.406,Z 228.572,A -85,B 0,C 180,E1 -579.127,E2 -579.127} C_VEL
LIN {X 0,Y 601.419,Z 228.567,A -85,B 0,C 180,E1 -581.766,E2 -581.766} C_VEL
LIN {X 0,Y 601.4,Z 228.577,A -85,B 0,C 180,E1 -584.533,E2 -584.533} C_VEL
LIN {X 0,Y 601.366,Z 228.574,A -85,B 0,C 180,E1 -587.414,E2 -587.414} C_VEL
LIN {X 0,Y 601.401,Z 228.572,A -85,B 0,C 180,E1 -590.004,E2 -590.004} C_VEL
LIN {X 0,Y 601.437,Z 228.565,A -85,B 0,C 180,E1 -592.618,E2 -592.618} C_VEL
LIN {X 0,Y 601.38,Z 228.572,A -85,B 0,C 180,E1 -594.245,E2 -594.245} C_VEL
LIN {X 0,Y 601.393,Z 229.253,A -85,B 0,C 180,E1 -595.067,E2 -595.067} C_VEL
LIN {X 0,Y 601.413,Z 233.392,A -85,B 0,C 180,E1 -597.483,E2 -597.483} C_VEL
LIN {X 0,Y 601.386,Z 238.84,A -85,B 0,C 180,E1 -600.605,E2 -600.605} C_VEL
LIN {X 0,Y 601.374,Z 242.891,A -85,B 0,C 180,E1 -602.885,E2 -602.885} C_VEL
LIN {X 0,Y 601.37,Z 248.42,A -85,B 0,C 180,E1 -605.856,E2 -605.856} C_VEL
LIN {X 0,Y 601.333,Z 252.567,A -85,B 0,C 180,E1 -608.038,E2 -608.038} C_VEL
LIN {X 0,Y 601.331,Z 256.714,A -85,B 0,C 180,E1 -610.188,E2 -610.188} C_VEL
LIN {X 0,Y 601.359,Z 262.243,A -85,B 0,C 180,E1 -613.012,E2 -613.012} C_VEL
LIN {X 0,Y 601.336,Z 268.073,A -85,B 0,C 180,E1 -615.942,E2 -615.942} C_VEL
LIN {X 0,Y 601.339,Z 272.526,A -85,B 0,C 180,E1 -618.155,E2 -618.155} C_VEL
LIN {X 0,Y 601.601,Z 277.391,A -85,B 0,C 180,E1 -618.268,E2 -618.268} C_VEL
LIN {X 0,Y 601.563,Z 289.681,A -85,B 0,C 180,E1 -618.583,E2 -618.583} C_VEL
LIN {X 0,Y 601.546,Z 302.829,A -85,B 0,C 180,E1 -619.073,E2 -619.073} C_VEL
LIN {X 0,Y 601.477,Z 314.514,A -85,B 0,C 180,E1 -619.651,E2 -619.651} C_VEL
LIN {X 0,Y 601.458,Z 325.31,A -85,B 0,C 180,E1 -620.33,E2 -620.33} C_VEL
LIN {X 0,Y 601.435,Z 335.085,A -85,B 0,C 180,E1 -621.093,E2 -621.093} C_VEL
LIN {X 0,Y 601.407,Z 343.981,A -85,B 0,C 180,E1 -621.939,E2 -621.939} C_VEL
LIN {X 0,Y 601.407,Z 352.667,A -85,B 0,C 180,E1 -622.952,E2 -622.952} C_VEL
LIN {X 0,Y 601.361,Z 359.597,A -85,B 0,C 180,E1 -623.962,E2 -623.962} C_VEL
LIN {X 0,Y 601.345,Z 365.149,A -85,B 0,C 180,E1 -624.971,E2 -624.971} C_VEL
LIN {X 0,Y 601.346,Z 369.511,A -85,B 0,C 180,E1 -625.979,E2 -625.979} C_VEL
LIN {X 0,Y 601.344,Z 371.815,A -85,B 0,C 180,E1 -626.65,E2 -626.65} C_VEL
LIN {X 0,Y 601.324,Z 373.693,A -85,B 0,C 180,E1 -627.32,E2 -627.32} C_VEL
LIN {X 0,Y 601.341,Z 375.127,A -85,B 0,C 180,E1 -627.991,E2 -627.991} C_VEL
LIN {X 0,Y 601.339,Z 376.753,A -85,B 0,C 180,E1 -629.33,E2 -629.33} C_VEL
LIN {X 0,Y 601.335,Z 376.996,A -85,B 0,C 180,E1 -630,E2 -630} C_VEL
LIN {X 0,Y 601.339,Z 376.815,A -85,B 0,C 180,E1 -630.67,E2 -630.67} C_VEL
LIN {X 0,Y 601.34,Z 375.275,A -85,B 0,C 180,E1 -632.009,E2 -632.009} C_VEL
LIN {X 0,Y 601.326,Z 373.916,A -85,B 0,C 180,E1 -632.68,E2 -632.68} C_VEL
LIN {X 0,Y 601.368,Z 371.04,A -85,B 0,C 180,E1 -633.685,E2 -633.685} C_VEL
LIN {X 0,Y 601.337,Z 367.14,A -85,B 0,C 180,E1 -634.693,E2 -634.693} C_VEL
LIN {X 0,Y 601.373,Z 362.109,A -85,B 0,C 180,E1 -635.701,E2 -635.701} C_VEL
LIN {X 0,Y 601.383,Z 355.791,A -85,B 0,C 180,E1 -636.711,E2 -636.711} C_VEL
LIN {X 0,Y 601.396,Z 347.873,A -85,B 0,C 180,E1 -637.723,E2 -637.723} C_VEL
LIN {X 0,Y 601.437,Z 338.029,A -85,B 0,C 180,E1 -638.738,E2 -638.738} C_VEL
LIN {X 0,Y 601.448,Z 327.707,A -85,B 0,C 180,E1 -639.585,E2 -639.585} C_VEL
LIN {X 0,Y 601.479,Z 316.087,A -85,B 0,C 180,E1 -640.349,E2 -640.349} C_VEL
LIN {X 0,Y 601.524,Z 304.195,A -85,B 0,C 180,E1 -640.959,E2 -640.959} C_VEL
LIN {X 0,Y 601.549,Z 291.243,A -85,B 0,C 180,E1 -641.456,E2 -641.456} C_VEL
LIN {X 0,Y 601.606,Z 278.616,A -85,B 0,C 180,E1 -641.797,E2 -641.797} C_VEL
LIN {X 0,Y 601.34,Z 272.534,A -85,B 0,C 180,E1 -641.93,E2 -641.93} C_VEL
LIN {X 0,Y 601.345,Z 266.57,A -85,B 0,C 180,E1 -644.899,E2 -644.899} C_VEL
LIN {X 0,Y 601.333,Z 261.038,A -85,B 0,C 180,E1 -647.69,E2 -647.69} C_VEL
LIN {X 0,Y 601.346,Z 255.505,A -85,B 0,C 180,E1 -650.525,E2 -650.525} C_VEL
LIN {X 0,Y 601.361,Z 249.972,A -85,B 0,C 180,E1 -653.413,E2 -653.413} C_VEL
LIN {X 0,Y 601.357,Z 244.439,A -85,B 0,C 180,E1 -656.366,E2 -656.366} C_VEL
LIN {X 0,Y 601.371,Z 240.08,A -85,B 0,C 180,E1 -658.777,E2 -658.777} C_VEL
LIN {X 0,Y 601.339,Z 235.417,A -85,B 0,C 180,E1 -661.442,E2 -661.442} C_VEL
LIN {X 0,Y 601.403,Z 231.106,A -85,B 0,C 180,E1 -663.931,E2 -663.931} C_VEL
LIN {X 0,Y 601.384,Z 229.11,A -85,B 0,C 180,E1 -665.11,E2 -665.11} C_VEL
LIN {X 0,Y 601.39,Z 228.572,A -85,B 0,C 180,E1 -665.755,E2 -665.755} C_VEL
LIN {X 0,Y 601.433,Z 228.569,A -85,B 0,C 180,E1 -668.471,E2 -668.471} C_VEL
LIN {X 0,Y 601.399,Z 228.57,A -85,B 0,C 180,E1 -670.876,E2 -670.876} C_VEL
LIN {X 0,Y 601.406,Z 228.572,A -85,B 0,C 180,E1 -673.589,E2 -673.589} C_VEL
LIN {X 0,Y 601.406,Z 228.568,A -85,B 0,C 180,E1 -676.43,E2 -676.43} C_VEL
LIN {X 0,Y 601.414,Z 228.572,A -85,B 0,C 180,E1 -679.125,E2 -679.125} C_VEL
LIN {X 0,Y 601.418,Z 228.567,A -85,B 0,C 180,E1 -681.732,E2 -681.732} C_VEL
LIN {X 0,Y 601.395,Z 228.575,A -85,B 0,C 180,E1 -684.246,E2 -684.246} C_VEL
LIN {X 0,Y 601.411,Z 228.567,A -85,B 0,C 180,E1 -686.685,E2 -686.685} C_VEL
LIN {X 0,Y 601.394,Z 228.575,A -85,B 0,C 180,E1 -689.056,E2 -689.056} C_VEL
LIN {X 0,Y 601.429,Z 228.567,A -85,B 0,C 180,E1 -691.373,E2 -691.373} C_VEL
LIN {X 0,Y 601.403,Z 228.569,A -85,B 0,C 180,E1 -693.636,E2 -693.636} C_VEL
LIN {X 0,Y 601.459,Z 228.566,A -85,B 0,C 180,E1 -695.86,E2 -695.86} C_VEL
LIN {X 0,Y 601.404,Z 228.568,A -85,B 0,C 180,E1 -698.76,E2 -698.76} C_VEL
LIN {X 0,Y 601.381,Z 228.573,A -85,B 0,C 180,E1 -701.607,E2 -701.607} C_VEL
LIN {X 0,Y 601.4,Z 228.573,A -85,B 0,C 180,E1 -704.408,E2 -704.408} C_VEL
LIN {X 0,Y 601.412,Z 228.567,A -85,B 0,C 180,E1 -707.172,E2 -707.172} C_VEL
LIN {X 0,Y 601.429,Z 228.571,A -85,B 0,C 180,E1 -709.905,E2 -709.905} C_VEL
LIN {X 0,Y 601.439,Z 228.565,A -85,B 0,C 180,E1 -712.615,E2 -712.615} C_VEL
LIN {X 0,Y 601.392,Z 228.572,A -85,B 0,C 180,E1 -715.308,E2 -715.308} C_VEL
LIN {X 0,Y 601.401,Z 228.571,A -85,B 0,C 180,E1 -717.991,E2 -717.991} C_VEL
LIN {X 0,Y 601.445,Z 228.564,A -85,B 0,C 180,E1 -720.669,E2 -720.669} C_VEL
LIN {X 0,Y 601.429,Z 228.571,A -85,B 0,C 180,E1 -723.35,E2 -723.35} C_VEL
LIN {X 0,Y 601.404,Z 228.568,A -85,B 0,C 180,E1 -726.037,E2 -726.037} C_VEL
LIN {X 0,Y 601.414,Z 228.573,A -85,B 0,C 180,E1 -728.738,E2 -728.738} C_VEL
LIN {X 0,Y 601.398,Z 228.57,A -85,B 0,C 180,E1 -731.459,E2 -731.459} C_VEL
LIN {X 0,Y 601.418,Z 228.568,A -85,B 0,C 180,E1 -734.206,E2 -734.206} C_VEL
LIN {X 0,Y 601.415,Z 228.572,A -85,B 0,C 180,E1 -736.986,E2 -736.986} C_VEL
LIN {X 0,Y 601.405,Z 228.568,A -85,B 0,C 180,E1 -739.81,E2 -739.81} C_VEL
LIN {X 0,Y 601.412,Z 228.57,A -85,B 0,C 180,E1 -742.683,E2 -742.683} C_VEL
LIN {X 0,Y 601.377,Z 228.571,A -85,B 0,C 180,E1 -744.88,E2 -744.88} C_VEL
LIN {X 0,Y 601.403,Z 228.575,A -85,B 0,C 180,E1 -747.359,E2 -747.359} C_VEL
LIN {X 0,Y 601.405,Z 228.568,A -85,B 0,C 180,E1 -750.165,E2 -750.165} C_VEL
LIN {X 0,Y 601.422,Z 228.572,A -85,B 0,C 180,E1 -752.715,E2 -752.715} C_VEL
LIN {X 0,Y 601.39,Z 228.57,A -85,B 0,C 180,E1 -755.111,E2 -755.111} C_VEL
LIN {X 0,Y 601.431,Z 228.568,A -85,B 0,C 180,E1 -757.419,E2 -757.419} C_VEL
LIN {X 0,Y 601.376,Z 228.573,A -85,B 0,C 180,E1 -759.998,E2 -759.998} C_VEL
LIN {X 0,Y 601.388,Z 228.575,A -85,B 0,C 180,E1 -762.673,E2 -762.673} C_VEL
LIN {X 0,Y 601.401,Z 228.569,A -85,B 0,C 180,E1 -765.479,E2 -765.479} C_VEL
LIN {X 0,Y 601.422,Z 228.568,A -85,B 0,C 180,E1 -768.407,E2 -768.407} C_VEL
LIN {X 0,Y 601.401,Z 228.57,A -85,B 0,C 180,E1 -770.872,E2 -770.872} C_VEL
LIN {X 0,Y 601.396,Z 228.575,A -85,B 0,C 180,E1 -773.416,E2 -773.416} C_VEL
LIN {X 0,Y 601.398,Z 228.633,A -85,B 0,C 180,E1 -774.332,E2 -774.332} C_VEL
LIN {X 0,Y 601.504,Z 235.01,A -85,B 0,C 180,E1 -776.691,E2 -776.691} C_VEL
LIN {X 0,Y 601.473,Z 242.89,A -85,B 0,C 180,E1 -779.45,E2 -779.45} C_VEL
LIN {X 0,Y 601.425,Z 250.751,A -85,B 0,C 180,E1 -782.133,E2 -782.133} C_VEL
LIN {X 0,Y 601.414,Z 259.656,A -85,B 0,C 180,E1 -785.122,E2 -785.122} C_VEL
LIN {X 0,Y 601.419,Z 266.572,A -85,B 0,C 180,E1 -787.395,E2 -787.395} C_VEL
LIN {X 0,Y 601.413,Z 275.239,A -85,B 0,C 180,E1 -790.191,E2 -790.191} C_VEL
LIN {X 0,Y 601.376,Z 284.143,A -85,B 0,C 180,E1 -793.012,E2 -793.012} C_VEL
LIN {X 0,Y 601.355,Z 293.048,A -85,B 0,C 180,E1 -795.793,E2 -795.793} C_VEL
LIN {X 0,Y 601.371,Z 300.491,A -85,B 0,C 180,E1 -798.092,E2 -798.092} C_VEL
LIN {X 0,Y 601.607,Z 307.506,A -85,B 0,C 180,E1 -798.225,E2 -798.225} C_VEL
LIN {X 0,Y 601.555,Z 319.876,A -85,B 0,C 180,E1 -798.544,E2 -798.544} C_VEL
LIN {X 0,Y 601.492,Z 332.863,A -85,B 0,C 180,E1 -799.028,E2 -799.028} C_VEL
LIN {X 0,Y 601.449,Z 345.325,A -85,B 0,C 180,E1 -799.65,E2 -799.65} C_VEL
LIN {X 0,Y 601.464,Z 355.93,A -85,B 0,C 180,E1 -800.33,E2 -800.33} C_VEL
LIN {X 0,Y 601.435,Z 365.598,A -85,B 0,C 180,E1 -801.093,E2 -801.093} C_VEL
LIN {X 0,Y 601.407,Z 374.412,A -85,B 0,C 180,E1 -801.939,E2 -801.939} C_VEL
LIN {X 0,Y 601.388,Z 381.69,A -85,B 0,C 180,E1 -802.783,E2 -802.783} C_VEL
LIN {X 0,Y 601.375,Z 388.773,A -85,B 0,C 180,E1 -803.782,E2 -803.782} C_VEL
LIN {X 0,Y 601.373,Z 393.68,A -85,B 0,C 180,E1 -804.635,E2 -804.635} C_VEL
LIN {X 0,Y 601.354,Z 398.371,A -85,B 0,C 180,E1 -805.643,E2 -805.643} C_VEL
LIN {X 0,Y 601.344,Z 401.956,A -85,B 0,C 180,E1 -806.65,E2 -806.65} C_VEL
LIN {X 0,Y 601.325,Z 403.809,A -85,B 0,C 180,E1 -807.32,E2 -807.32} C_VEL
LIN {X 0,Y 601.343,Z 405.201,A -85,B 0,C 180,E1 -807.991,E2 -807.991} C_VEL
LIN {X 0,Y 601.339,Z 406.784,A -85,B 0,C 180,E1 -809.33,E2 -809.33} C_VEL
LIN {X 0,Y 601.335,Z 407,A -85,B 0,C 180,E1 -810,E2 -810} C_VEL
LIN {X 0,Y 601.347,Z 406.184,A -85,B 0,C 180,E1 -811.339,E2 -811.339} C_VEL
LIN {X 0,Y 601.343,Z 405.202,A -85,B 0,C 180,E1 -812.009,E2 -812.009} C_VEL
LIN {X 0,Y 601.325,Z 403.809,A -85,B 0,C 180,E1 -812.68,E2 -812.68} C_VEL
LIN {X 0,Y 601.368,Z 400.896,A -85,B 0,C 180,E1 -813.685,E2 -813.685} C_VEL
LIN {X 0,Y 601.336,Z 396.95,A -85,B 0,C 180,E1 -814.693,E2 -814.693} C_VEL
LIN {X 0,Y 601.373,Z 390.877,A -85,B 0,C 180,E1 -815.869,E2 -815.869} C_VEL
LIN {X 0,Y 601.382,Z 384.236,A -85,B 0,C 180,E1 -816.88,E2 -816.88} C_VEL
LIN {X 0,Y 601.4,Z 375.99,A -85,B 0,C 180,E1 -817.892,E2 -817.892} C_VEL
LIN {X 0,Y 601.436,Z 367.537,A -85,B 0,C 180,E1 -818.738,E2 -818.738} C_VEL
LIN {X 0,Y 601.447,Z 357.093,A -85,B 0,C 180,E1 -819.585,E2 -819.585} C_VEL
LIN {X 0,Y 601.473,Z 346.758,A -85,B 0,C 180,E1 -820.264,E2 -820.264} C_VEL
LIN {X 0,Y 601.481,Z 335.25,A -85,B 0,C 180,E1 -820.868,E2 -820.868} C_VEL
LIN {X 0,Y 601.526,Z 322.34,A -85,B 0,C 180,E1 -821.375,E2 -821.375} C_VEL
LIN {X 0,Y 601.611,Z 309.439,A -85,B 0,C 180,E1 -821.732,E2 -821.732} C_VEL
LIN {X 0,Y 601.501,Z 301.615,A -85,B 0,C 180,E1 -821.884,E2 -821.884} C_VEL
LIN {X 0,Y 601.342,Z 300.422,A -85,B 0,C 180,E1 -821.93,E2 -821.93} C_VEL
LIN {X 0,Y 601.352,Z 291.935,A -85,B 0,C 180,E1 -824.553,E2 -824.553} C_VEL
LIN {X 0,Y 601.394,Z 283.031,A -85,B 0,C 180,E1 -827.337,E2 -827.337} C_VEL
LIN {X 0,Y 601.394,Z 274.126,A -85,B 0,C 180,E1 -830.166,E2 -830.166} C_VEL
LIN {X 0,Y 601.413,Z 266.335,A -85,B 0,C 180,E1 -832.683,E2 -832.683} C_VEL
LIN {X 0,Y 601.41,Z 258.543,A -85,B 0,C 180,E1 -835.248,E2 -835.248} C_VEL
LIN {X 0,Y 601.425,Z 250.751,A -85,B 0,C 180,E1 -837.867,E2 -837.867} C_VEL
LIN {X 0,Y 601.473,Z 242.89,A -85,B 0,C 180,E1 -840.55,E2 -840.55} C_VEL
LIN {X 0,Y 601.503,Z 235.011,A -85,B 0,C 180,E1 -843.309,E2 -843.309} C_VEL
LIN {X 0,Y 601.403,Z 228.573,A -85,B 0,C 180,E1 -845.711,E2 -845.711} C_VEL
LIN {X 0,Y 601.406,Z 228.575,A -85,B 0,C 180,E1 -848.468,E2 -848.468} C_VEL
LIN {X 0,Y 601.412,Z 228.569,A -85,B 0,C 180,E1 -850.875,E2 -850.875} C_VEL
LIN {X 0,Y 601.43,Z 228.571,A -85,B 0,C 180,E1 -853.586,E2 -853.586} C_VEL
LIN {X 0,Y 601.431,Z 228.565,A -85,B 0,C 180,E1 -856.427,E2 -856.427} C_VEL
LIN {X 0,Y 601.401,Z 228.572,A -85,B 0,C 180,E1 -859.124,E2 -859.124} C_VEL
LIN {X 0,Y 601.367,Z 228.574,A -85,B 0,C 180,E1 -861.728,E2 -861.728} C_VEL
LIN {X 0,Y 601.389,Z 228.574,A -85,B 0,C 180,E1 -864.245,E2 -864.245} C_VEL
LIN {X 0,Y 601.43,Z 228.565,A -85,B 0,C 180,E1 -866.687,E2 -866.687} C_VEL
LIN {X 0,Y 601.424,Z 228.573,A -85,B 0,C 180,E1 -869.058,E2 -869.058} C_VEL
LIN {X 0,Y 601.408,Z 228.569,A -85,B 0,C 180,E1 -871.372,E2 -871.372} C_VEL
LIN {X 0,Y 601.408,Z 228.573,A -85,B 0,C 180,E1 -874.134,E2 -874.134} C_VEL
LIN {X 0,Y 601.383,Z 228.571,A -85,B 0,C 180,E1 -876.588,E2 -876.588} C_VEL
LIN {X 0,Y 601.433,Z 228.572,A -85,B 0,C 180,E1 -879.478,E2 -879.478} C_VEL
LIN {X 0,Y 601.401,Z 228.57,A -85,B 0,C 180,E1 -882.312,E2 -882.312} C_VEL
LIN {X 0,Y 601.413,Z 228.573,A -85,B 0,C 180,E1 -884.409,E2 -884.409} C_VEL
LIN {X 0,Y 601.395,Z 228.569,A -85,B 0,C 180,E1 -887.171,E2 -887.171} C_VEL
LIN {X 0,Y 601.391,Z 228.575,A -85,B 0,C 180,E1 -889.904,E2 -889.904} C_VEL
LIN {X 0,Y 601.399,Z 228.57,A -85,B 0,C 180,E1 -892.614,E2 -892.614} C_VEL
LIN {X 0,Y 601.426,Z 228.567,A -85,B 0,C 180,E1 -895.308,E2 -895.308} C_VEL
LIN {X 0,Y 601.429,Z 228.569,A -85,B 0,C 180,E1 -897.991,E2 -897.991} C_VEL
LIN {X 0,Y 601.424,Z 228.566,A -85,B 0,C 180,E1 -900.67,E2 -900.67} C_VEL
LIN {X 0,Y 601.416,Z 228.574,A -85,B 0,C 180,E1 -903.35,E2 -903.35} C_VEL
LIN {X 0,Y 601.382,Z 228.571,A -85,B 0,C 180,E1 -906.037,E2 -906.037} C_VEL
LIN {X 0,Y 601.441,Z 228.569,A -85,B 0,C 180,E1 -908.738,E2 -908.738} C_VEL
LIN {X 0,Y 601.441,Z 228.565,A -85,B 0,C 180,E1 -911.458,E2 -911.458} C_VEL
LIN {X 0,Y 601.407,Z 228.571,A -85,B 0,C 180,E1 -912.357,E2 -912.357} C_VEL
LIN {X 0,Y 600.736,Z 228.652,A -85,B 0,C 180,E1 -912.917,E2 -912.917} C_VEL
LIN {X 0,Y 597.879,Z 229.014,A -85,B 0,C 180,E1 -913.824,E2 -913.824} C_VEL
LIN {X 0,Y 595.466,Z 229.313,A -85,B 0,C 180,E1 -914.554,E2 -914.554} C_VEL
LIN {X 0,Y 594.428,Z 229.441,A -85,B 0,C 180,E1 -915.118,E2 -915.118} C_VEL
LIN {X 0,Y 594.342,Z 229.45,A -85,B 0,C 180,E1 -915.309,E2 -915.309} C_VEL
LIN {X 0,Y 594.325,Z 229.45,A -85,B 0,C 180,E1 -917.906,E2 -917.906} C_VEL
LIN {X 0,Y 594.407,Z 229.444,A -85,B 0,C 180,E1 -920.776,E2 -920.776} C_VEL
LIN {X 0,Y 594.38,Z 229.447,A -85,B 0,C 180,E1 -923.705,E2 -923.705} C_VEL
LIN {X 0,Y 594.387,Z 229.443,A -85,B 0,C 180,E1 -926.7,E2 -926.7} C_VEL
LIN {X 0,Y 594.379,Z 229.449,A -85,B 0,C 180,E1 -928.999,E2 -928.999} C_VEL
LIN {X 0,Y 594.367,Z 229.445,A -85,B 0,C 180,E1 -931.641,E2 -931.641} C_VEL
LIN {X 0,Y 594.368,Z 229.448,A -85,B 0,C 180,E1 -934.581,E2 -934.581} C_VEL
LIN {X 0,Y 594.389,Z 229.449,A -85,B 0,C 180,E1 -937.608,E2 -937.608} C_VEL
LIN {X 0,Y 594.37,Z 229.446,A -85,B 0,C 180,E1 -940.567,E2 -940.567} C_VEL
LIN {X 0,Y 594.353,Z 229.448,A -85,B 0,C 180,E1 -943.301,E2 -943.301} C_VEL
LIN {X 0,Y 594.336,Z 229.455,A -85,B 0,C 180,E1 -946.164,E2 -946.164} C_VEL
LIN {X 0,Y 594.368,Z 229.446,A -85,B 0,C 180,E1 -948.535,E2 -948.535} C_VEL
LIN {X 0,Y 594.381,Z 229.449,A -85,B 0,C 180,E1 -951.296,E2 -951.296} C_VEL
LIN {X 0,Y 594.355,Z 229.447,A -85,B 0,C 180,E1 -953.756,E2 -953.756} C_VEL
LIN {X 0,Y 594.307,Z 229.487,A -85,B 0,C 180,E1 -954.683,E2 -954.683} C_VEL
LIN {X 0,Y 594.339,Z 233.529,A -85,B 0,C 180,E1 -957.095,E2 -957.095} C_VEL
LIN {X 0,Y 594.312,Z 237.981,A -85,B 0,C 180,E1 -959.685,E2 -959.685} C_VEL
LIN {X 0,Y 594.32,Z 241.622,A -85,B 0,C 180,E1 -961.77,E2 -961.77} C_VEL
LIN {X 0,Y 594.282,Z 247.039,A -85,B 0,C 180,E1 -964.803,E2 -964.803} C_VEL
LIN {X 0,Y 594.267,Z 252.568,A -85,B 0,C 180,E1 -967.763,E2 -967.763} C_VEL
LIN {X 0,Y 594.242,Z 256.715,A -85,B 0,C 180,E1 -969.942,E2 -969.942} C_VEL
LIN {X 0,Y 594.256,Z 262.245,A -85,B 0,C 180,E1 -972.803,E2 -972.803} C_VEL
LIN {X 0,Y 594.255,Z 267.774,A -85,B 0,C 180,E1 -975.62,E2 -975.62} C_VEL
LIN {X 0,Y 594.268,Z 272.527,A -85,B 0,C 180,E1 -978.012,E2 -978.012} C_VEL
LIN {X 0,Y 594.656,Z 277.419,A -85,B 0,C 180,E1 -978.129,E2 -978.129} C_VEL
LIN {X 0,Y 594.61,Z 289.78,A -85,B 0,C 180,E1 -978.45,E2 -978.45} C_VEL
LIN {X 0,Y 594.561,Z 302.843,A -85,B 0,C 180,E1 -978.943,E2 -978.943} C_VEL
LIN {X 0,Y 594.489,Z 314.526,A -85,B 0,C 180,E1 -979.528,E2 -979.528} C_VEL
LIN {X 0,Y 594.438,Z 325.316,A -85,B 0,C 180,E1 -980.215,E2 -980.215} C_VEL
LIN {X 0,Y 594.404,Z 335.092,A -85,B 0,C 180,E1 -980.987,E2 -980.987} C_VEL
LIN {X 0,Y 594.366,Z 343.986,A -85,B 0,C 180,E1 -981.843,E2 -981.843} C_VEL
LIN {X 0,Y 594.345,Z 352.672,A -85,B 0,C 180,E1 -982.868,E2 -982.868} C_VEL
LIN {X 0,Y 594.29,Z 359.6,A -85,B 0,C 180,E1 -983.89,E2 -983.89} C_VEL
LIN {X 0,Y 594.254,Z 365.152,A -85,B 0,C 180,E1 -984.911,E2 -984.911} C_VEL
LIN {X 0,Y 594.262,Z 369.514,A -85,B 0,C 180,E1 -985.931,E2 -985.931} C_VEL
LIN {X 0,Y 594.267,Z 371.817,A -85,B 0,C 180,E1 -986.61,E2 -986.61} C_VEL
LIN {X 0,Y 594.225,Z 373.695,A -85,B 0,C 180,E1 -987.288,E2 -987.288} C_VEL
LIN {X 0,Y 594.24,Z 375.127,A -85,B 0,C 180,E1 -987.967,E2 -987.967} C_VEL
LIN {X 0,Y 594.24,Z 376.753,A -85,B 0,C 180,E1 -989.322,E2 -989.322} C_VEL
LIN {X 0,Y 594.236,Z 376.996,A -85,B 0,C 180,E1 -990,E2 -990} C_VEL
LIN {X 0,Y 594.239,Z 376.815,A -85,B 0,C 180,E1 -990.678,E2 -990.678} C_VEL
LIN {X 0,Y 594.239,Z 375.275,A -85,B 0,C 180,E1 -992.033,E2 -992.033} C_VEL
LIN {X 0,Y 594.227,Z 373.914,A -85,B 0,C 180,E1 -992.712,E2 -992.712} C_VEL
LIN {X 0,Y 594.289,Z 371.038,A -85,B 0,C 180,E1 -993.729,E2 -993.729} C_VEL
LIN {X 0,Y 594.241,Z 367.138,A -85,B 0,C 180,E1 -994.749,E2 -994.749} C_VEL
LIN {X 0,Y 594.299,Z 362.106,A -85,B 0,C 180,E1 -995.769,E2 -995.769} C_VEL
LIN {X 0,Y 594.316,Z 355.787,A -85,B 0,C 180,E1 -996.791,E2 -996.791} C_VEL
LIN {X 0,Y 594.346,Z 347.869,A -85,B 0,C 180,E1 -997.816,E2 -997.816} C_VEL
LIN {X 0,Y 594.381,Z 338.022,A -85,B 0,C 180,E1 -998.842,E2 -998.842} C_VEL
LIN {X 0,Y 594.429,Z 327.701,A -85,B 0,C 180,E1 -999.7,E2 -999.7} C_VEL
LIN {X 0,Y 594.473,Z 317.495,A -85,B 0,C 180,E1 -1000.387,E2 -1000.387} C_VEL
LIN {X 0,Y 594.554,Z 305.675,A -85,B 0,C 180,E1 -1001.021,E2 -1001.021} C_VEL
LIN {X 0,Y 594.617,Z 293.786,A -85,B 0,C 180,E1 -1001.506,E2 -1001.506} C_VEL
LIN {X 0,Y 594.65,Z 281.337,A -85,B 0,C 180,E1 -1001.872,E2 -1001.872} C_VEL
LIN {X 0,Y 594.49,Z 274.171,A -85,B 0,C 180,E1 -1002.026,E2 -1002.026} C_VEL
LIN {X 0,Y 594.256,Z 272.533,A -85,B 0,C 180,E1 -1002.075,E2 -1002.075} C_VEL
LIN {X 0,Y 594.263,Z 266.569,A -85,B 0,C 180,E1 -1005.081,E2 -1005.081} C_VEL
LIN {X 0,Y 594.258,Z 262.42,A -85,B 0,C 180,E1 -1007.197,E2 -1007.197} C_VEL
LIN {X 0,Y 594.243,Z 256.887,A -85,B 0,C 180,E1 -1010.059,E2 -1010.059} C_VEL
LIN {X 0,Y 594.308,Z 251.822,A -85,B 0,C 180,E1 -1012.721,E2 -1012.721} C_VEL
LIN {X 0,Y 594.284,Z 247.205,A -85,B 0,C 180,E1 -1015.197,E2 -1015.197} C_VEL
LIN {X 0,Y 594.32,Z 241.781,A -85,B 0,C 180,E1 -1018.23,E2 -1018.23} C_VEL
LIN {X 0,Y 594.288,Z 237.715,A -85,B 0,C 180,E1 -1020.565,E2 -1020.565} C_VEL
LIN {X 0,Y 594.331,Z 233.6,A -85,B 0,C 180,E1 -1022.953,E2 -1022.953} C_VEL
LIN {X 0,Y 594.313,Z 229.479,A -85,B 0,C 180,E1 -1025.412,E2 -1025.412} C_VEL
LIN {X 0,Y 594.389,Z 229.442,A -85,B 0,C 180,E1 -1027.941,E2 -1027.941} C_VEL
LIN {X 0,Y 594.366,Z 229.447,A -85,B 0,C 180,E1 -1030.82,E2 -1030.82} C_VEL
LIN {X 0,Y 594.341,Z 229.449,A -85,B 0,C 180,E1 -1033.302,E2 -1033.302} C_VEL
LIN {X 0,Y 594.345,Z 229.448,A -85,B 0,C 180,E1 -1036.163,E2 -1036.163} C_VEL
LIN {X 0,Y 594.377,Z 229.446,A -85,B 0,C 180,E1 -1038.536,E2 -1038.536} C_VEL
LIN {X 0,Y 594.377,Z 229.444,A -85,B 0,C 180,E1 -1041.297,E2 -1041.297} C_VEL
LIN {X 0,Y 594.364,Z 229.448,A -85,B 0,C 180,E1 -1043.756,E2 -1043.756} C_VEL
LIN {X 0,Y 594.356,Z 229.448,A -85,B 0,C 180,E1 -1046.237,E2 -1046.237} C_VEL
LIN {X 0,Y 594.358,Z 229.447,A -85,B 0,C 180,E1 -1048.649,E2 -1048.649} C_VEL
LIN {X 0,Y 594.372,Z 229.444,A -85,B 0,C 180,E1 -1051.773,E2 -1051.773} C_VEL
LIN {X 0,Y 594.376,Z 229.447,A -85,B 0,C 180,E1 -1054.056,E2 -1054.056} C_VEL
LIN {X 0,Y 594.38,Z 229.448,A -85,B 0,C 180,E1 -1056.295,E2 -1056.295} C_VEL
LIN {X 0,Y 594.41,Z 229.443,A -85,B 0,C 180,E1 -1059.225,E2 -1059.225} C_VEL
LIN {X 0,Y 594.326,Z 229.45,A -85,B 0,C 180,E1 -1062.094,E2 -1062.094} C_VEL
LIN {X 0,Y 594.348,Z 229.449,A -85,B 0,C 180,E1 -1064.218,E2 -1064.218} C_VEL
LIN {X 0,Y 594.36,Z 229.446,A -85,B 0,C 180,E1 -1067.017,E2 -1067.017} C_VEL
LIN {X 0,Y 594.389,Z 229.45,A -85,B 0,C 180,E1 -1069.784,E2 -1069.784} C_VEL
LIN {X 0,Y 594.391,Z 229.442,A -85,B 0,C 180,E1 -1072.527,E2 -1072.527} C_VEL
LIN {X 0,Y 594.367,Z 229.448,A -85,B 0,C 180,E1 -1075.252,E2 -1075.252} C_VEL
LIN {X 0,Y 594.373,Z 229.447,A -85,B 0,C 180,E1 -1077.967,E2 -1077.967} C_VEL
LIN {X 0,Y 594.417,Z 229.439,A -85,B 0,C 180,E1 -1080.677,E2 -1080.677} C_VEL
LIN {X 0,Y 594.38,Z 229.45,A -85,B 0,C 180,E1 -1083.389,E2 -1083.389} C_VEL
LIN {X 0,Y 594.359,Z 229.446,A -85,B 0,C 180,E1 -1086.109,E2 -1086.109} C_VEL
LIN {X 0,Y 594.376,Z 229.448,A -85,B 0,C 180,E1 -1088.842,E2 -1088.842} C_VEL
LIN {X 0,Y 594.371,Z 229.446,A -85,B 0,C 180,E1 -1091.596,E2 -1091.596} C_VEL
LIN {X 0,Y 594.386,Z 229.443,A -85,B 0,C 180,E1 -1094.377,E2 -1094.377} C_VEL
LIN {X 0,Y 594.383,Z 229.45,A -85,B 0,C 180,E1 -1097.194,E2 -1097.194} C_VEL
LIN {X 0,Y 594.376,Z 229.445,A -85,B 0,C 180,E1 -1100.054,E2 -1100.054} C_VEL
LIN {X 0,Y 594.355,Z 229.447,A -85,B 0,C 180,E1 -1102.968,E2 -1102.968} C_VEL
LIN {X 0,Y 594.334,Z 229.45,A -85,B 0,C 180,E1 -1105.195,E2 -1105.195} C_VEL
LIN {X 0,Y 594.349,Z 229.454,A -85,B 0,C 180,E1 -1107.519,E2 -1107.519} C_VEL
LIN {X 0,Y 594.372,Z 229.445,A -85,B 0,C 180,E1 -1110.325,E2 -1110.325} C_VEL
LIN {X 0,Y 594.382,Z 229.446,A -85,B 0,C 180,E1 -1112.95,E2 -1112.95} C_VEL
LIN {X 0,Y 594.351,Z 229.448,A -85,B 0,C 180,E1 -1115.409,E2 -1115.409} C_VEL
LIN {X 0,Y 594.357,Z 229.45,A -85,B 0,C 180,E1 -1117.943,E2 -1117.943} C_VEL
LIN {X 0,Y 594.361,Z 229.449,A -85,B 0,C 180,E1 -1120.82,E2 -1120.82} C_VEL
LIN {X 0,Y 594.363,Z 229.446,A -85,B 0,C 180,E1 -1123.839,E2 -1123.839} C_VEL
LIN {X 0,Y 594.369,Z 229.447,A -85,B 0,C 180,E1 -1126.7,E2 -1126.7} C_VEL
LIN {X 0,Y 594.369,Z 229.449,A -85,B 0,C 180,E1 -1129.433,E2 -1129.433} C_VEL
LIN {X 0,Y 594.383,Z 229.444,A -85,B 0,C 180,E1 -1132.393,E2 -1132.393} C_VEL
LIN {X 0,Y 594.36,Z 229.463,A -85,B 0,C 180,E1 -1134.175,E2 -1134.175} C_VEL
LIN {X 0,Y 594.47,Z 233.893,A -85,B 0,C 180,E1 -1135.849,E2 -1135.849} C_VEL
LIN {X 0,Y 594.448,Z 240.8,A -85,B 0,C 180,E1 -1138.347,E2 -1138.347} C_VEL
LIN {X 0,Y 594.425,Z 248.541,A -85,B 0,C 180,E1 -1141.035,E2 -1141.035} C_VEL
LIN {X 0,Y 594.378,Z 255.2,A -85,B 0,C 180,E1 -1143.3,E2 -1143.3} C_VEL
LIN {X 0,Y 594.41,Z 263.01,A -85,B 0,C 180,E1 -1145.931,E2 -1145.931} C_VEL
LIN {X 0,Y 594.388,Z 270.786,A -85,B 0,C 180,E1 -1148.497,E2 -1148.497} C_VEL
LIN {X 0,Y 594.328,Z 279.691,A -85,B 0,C 180,E1 -1151.381,E2 -1151.381} C_VEL
LIN {X 0,Y 594.302,Z 288.595,A -85,B 0,C 180,E1 -1154.217,E2 -1154.217} C_VEL
LIN {X 0,Y 594.276,Z 297.5,A -85,B 0,C 180,E1 -1157.015,E2 -1157.015} C_VEL
LIN {X 0,Y 594.28,Z 300.491,A -85,B 0,C 180,E1 -1157.948,E2 -1157.948} C_VEL
LIN {X 0,Y 594.668,Z 305.224,A -85,B 0,C 180,E1 -1158.042,E2 -1158.042} C_VEL
LIN {X 0,Y 594.612,Z 318.493,A -85,B 0,C 180,E1 -1158.365,E2 -1158.365} C_VEL
LIN {X 0,Y 594.53,Z 330.675,A -85,B 0,C 180,E1 -1158.802,E2 -1158.802} C_VEL
LIN {X 0,Y 594.472,Z 342.208,A -85,B 0,C 180,E1 -1159.355,E2 -1159.355} C_VEL
LIN {X 0,Y 594.459,Z 353.476,A -85,B 0,C 180,E1 -1160.043,E2 -1160.043} C_VEL
LIN {X 0,Y 594.406,Z 363.646,A -85,B 0,C 180,E1 -1160.815,E2 -1160.815} C_VEL
LIN {X 0,Y 594.372,Z 372.786,A -85,B 0,C 180,E1 -1161.671,E2 -1161.671} C_VEL
LIN {X 0,Y 594.316,Z 381.69,A -85,B 0,C 180,E1 -1162.697,E2 -1162.697} C_VEL
LIN {X 0,Y 594.281,Z 388.168,A -85,B 0,C 180,E1 -1163.615,E2 -1163.615} C_VEL
LIN {X 0,Y 594.289,Z 393.68,A -85,B 0,C 180,E1 -1164.571,E2 -1164.571} C_VEL
LIN {X 0,Y 594.27,Z 398.371,A -85,B 0,C 180,E1 -1165.591,E2 -1165.591} C_VEL
LIN {X 0,Y 594.267,Z 401.956,A -85,B 0,C 180,E1 -1166.61,E2 -1166.61} C_VEL
LIN {X 0,Y 594.226,Z 403.809,A -85,B 0,C 180,E1 -1167.288,E2 -1167.288} C_VEL
LIN {X 0,Y 594.242,Z 405.201,A -85,B 0,C 180,E1 -1167.967,E2 -1167.967} C_VEL
LIN {X 0,Y 594.239,Z 406.784,A -85,B 0,C 180,E1 -1169.322,E2 -1169.322} C_VEL
LIN {X 0,Y 594.236,Z 407,A -85,B 0,C 180,E1 -1170,E2 -1170} C_VEL
LIN {X 0,Y 594.247,Z 406.185,A -85,B 0,C 180,E1 -1171.355,E2 -1171.355} C_VEL
LIN {X 0,Y 594.242,Z 405.202,A -85,B 0,C 180,E1 -1172.033,E2 -1172.033} C_VEL
LIN {X 0,Y 594.226,Z 403.81,A -85,B 0,C 180,E1 -1172.712,E2 -1172.712} C_VEL
LIN {X 0,Y 594.289,Z 400.896,A -85,B 0,C 180,E1 -1173.729,E2 -1173.729} C_VEL
LIN {X 0,Y 594.241,Z 396.95,A -85,B 0,C 180,E1 -1174.749,E2 -1174.749} C_VEL
LIN {X 0,Y 594.305,Z 390.878,A -85,B 0,C 180,E1 -1175.939,E2 -1175.939} C_VEL
LIN {X 0,Y 594.308,Z 384.236,A -85,B 0,C 180,E1 -1176.962,E2 -1176.962} C_VEL
LIN {X 0,Y 594.359,Z 375.99,A -85,B 0,C 180,E1 -1177.986,E2 -1177.986} C_VEL
LIN {X 0,Y 594.382,Z 367.538,A -85,B 0,C 180,E1 -1178.842,E2 -1178.842} C_VEL
LIN {X 0,Y 594.432,Z 357.094,A -85,B 0,C 180,E1 -1179.699,E2 -1179.699} C_VEL
LIN {X 0,Y 594.45,Z 346.759,A -85,B 0,C 180,E1 -1180.387,E2 -1180.387} C_VEL
LIN {X 0,Y 594.499,Z 334.78,A -85,B 0,C 180,E1 -1181.019,E2 -1181.019} C_VEL
LIN {X 0,Y 594.56,Z 322.495,A -85,B 0,C 180,E1 -1181.505,E2 -1181.505} C_VEL
LIN {X 0,Y 594.68,Z 309.437,A -85,B 0,C 180,E1 -1181.871,E2 -1181.871} C_VEL
LIN {X 0,Y 594.419,Z 301.614,A -85,B 0,C 180,E1 -1182.028,E2 -1182.028} C_VEL
LIN {X 0,Y 594.285,Z 300.422,A -85,B 0,C 180,E1 -1182.074,E2 -1182.074} C_VEL
LIN {X 0,Y 594.299,Z 291.935,A -85,B 0,C 180,E1 -1184.729,E2 -1184.729} C_VEL
LIN {X 0,Y 594.325,Z 283.031,A -85,B 0,C 180,E1 -1187.55,E2 -1187.55} C_VEL
LIN {X 0,Y 594.358,Z 274.126,A -85,B 0,C 180,E1 -1190.415,E2 -1190.415} C_VEL
LIN {X 0,Y 594.376,Z 266.335,A -85,B 0,C 180,E1 -1192.967,E2 -1192.967} C_VEL
LIN {X 0,Y 594.407,Z 258.543,A -85,B 0,C 180,E1 -1195.567,E2 -1195.567} C_VEL
LIN {X 0,Y 594.405,Z 250.705,A -85,B 0,C 180,E1 -1198.226,E2 -1198.226} C_VEL
LIN {X 0,Y 594.466,Z 242.806,A -85,B 0,C 180,E1 -1200.949,E2 -1200.949} C_VEL
LIN {X 0,Y 594.495,Z 234.96,A -85,B 0,C 180,E1 -1203.754,E2 -1203.754} C_VEL
LIN {X 0,Y 594.518,Z 230.568,A -85,B 0,C 180,E1 -1205.398,E2 -1205.398} C_VEL
LIN {X 0,Y 594.339,Z 229.453,A -85,B 0,C 180,E1 -1205.879,E2 -1205.879} C_VEL
LIN {X 0,Y 594.371,Z 229.446,A -85,B 0,C 180,E1 -1207.942,E2 -1207.942} C_VEL
LIN {X 0,Y 594.376,Z 229.446,A -85,B 0,C 180,E1 -1210.822,E2 -1210.822} C_VEL
LIN {X 0,Y 594.368,Z 229.447,A -85,B 0,C 180,E1 -1213.299,E2 -1213.299} C_VEL
LIN {X 0,Y 594.362,Z 229.446,A -85,B 0,C 180,E1 -1216.161,E2 -1216.161} C_VEL
LIN {X 0,Y 594.361,Z 229.449,A -85,B 0,C 180,E1 -1219.18,E2 -1219.18} C_VEL
LIN {X 0,Y 594.356,Z 229.45,A -85,B 0,C 180,E1 -1222.057,E2 -1222.057} C_VEL
LIN {X 0,Y 594.351,Z 229.447,A -85,B 0,C 180,E1 -1224.677,E2 -1224.677} C_VEL
LIN {X 0,Y 594.381,Z 229.446,A -85,B 0,C 180,E1 -1227.088,E2 -1227.088} C_VEL
LIN {X 0,Y 594.374,Z 229.445,A -85,B 0,C 180,E1 -1229.674,E2 -1229.674} C_VEL
LIN {X 0,Y 594.377,Z 229.451,A -85,B 0,C 180,E1 -1232.539,E2 -1232.539} C_VEL
LIN {X 0,Y 594.367,Z 229.446,A -85,B 0,C 180,E1 -1235.553,E2 -1235.553} C_VEL
LIN {X 0,Y 594.36,Z 229.446,A -85,B 0,C 180,E1 -1238.496,E2 -1238.496} C_VEL
LIN {X 0,Y 594.387,Z 229.447,A -85,B 0,C 180,E1 -1241.383,E2 -1241.383} C_VEL
LIN {X 0,Y 594.366,Z 229.448,A -85,B 0,C 180,E1 -1244.219,E2 -1244.219} C_VEL
LIN {X 0,Y 594.373,Z 229.451,A -85,B 0,C 180,E1 -1246.321,E2 -1246.321} C_VEL
LIN {X 0,Y 594.365,Z 229.446,A -85,B 0,C 180,E1 -1249.094,E2 -1249.094} C_VEL
LIN {X 0,Y 594.361,Z 229.448,A -85,B 0,C 180,E1 -1251.843,E2 -1251.843} C_VEL
LIN {X 0,Y 594.39,Z 229.446,A -85,B 0,C 180,E1 -1254.572,E2 -1254.572} C_VEL
LIN {X 0,Y 594.409,Z 229.44,A -85,B 0,C 180,E1 -1257.289,E2 -1257.289} C_VEL
LIN {X 0,Y 594.414,Z 229.446,A -85,B 0,C 180,E1 -1260,E2 -1260} C_VEL
LIN {X 0,Y 594.372,Z 229.444,A -85,B 0,C 180,E1 -1262.711,E2 -1262.711} C_VEL
LIN {X 0,Y 594.391,Z 229.445,A -85,B 0,C 180,E1 -1265.428,E2 -1265.428} C_VEL
LIN {X 0,Y 594.366,Z 229.447,A -85,B 0,C 180,E1 -1268.157,E2 -1268.157} C_VEL
LIN {X 0,Y 594.392,Z 229.442,A -85,B 0,C 180,E1 -1271.073,E2 -1271.073} C_VEL
LIN {X 0,Y 594.377,Z 229.451,A -85,B 0,C 180,E1 -1273.679,E2 -1273.679} C_VEL
LIN {X 0,Y 594.342,Z 229.45,A -85,B 0,C 180,E1 -1275.309,E2 -1275.309} C_VEL
LIN {X 0,Y 593.667,Z 229.535,A -85,B 0,C 180,E1 -1275.874,E2 -1275.874} C_VEL
LIN {X 0,Y 590.793,Z 229.893,A -85,B 0,C 180,E1 -1276.792,E2 -1276.792} C_VEL
LIN {X 0,Y 588.379,Z 230.193,A -85,B 0,C 180,E1 -1277.53,E2 -1277.53} C_VEL
LIN {X 0,Y 587.36,Z 230.318,A -85,B 0,C 180,E1 -1278.1,E2 -1278.1} C_VEL
LIN {X 0,Y 587.286,Z 230.328,A -85,B 0,C 180,E1 -1278.293,E2 -1278.293} C_VEL
LIN {X 0,Y 587.334,Z 230.322,A -85,B 0,C 180,E1 -1281.038,E2 -1281.038} C_VEL
LIN {X 0,Y 587.317,Z 230.323,A -85,B 0,C 180,E1 -1283.259,E2 -1283.259} C_VEL
LIN {X 0,Y 587.339,Z 230.326,A -85,B 0,C 180,E1 -1285.517,E2 -1285.517} C_VEL
LIN {X 0,Y 587.341,Z 230.323,A -85,B 0,C 180,E1 -1287.818,E2 -1287.818} C_VEL
LIN {X 0,Y 587.308,Z 230.327,A -85,B 0,C 180,E1 -1290.505,E2 -1290.505} C_VEL
LIN {X 0,Y 587.329,Z 230.323,A -85,B 0,C 180,E1 -1293.11,E2 -1293.11} C_VEL
LIN {X 0,Y 587.285,Z 230.334,A -85,B 0,C 180,E1 -1295.901,E2 -1295.901} C_VEL
LIN {X 0,Y 587.325,Z 230.322,A -85,B 0,C 180,E1 -1298.48,E2 -1298.48} C_VEL
LIN {X 0,Y 587.337,Z 230.328,A -85,B 0,C 180,E1 -1301.157,E2 -1301.157} C_VEL
LIN {X 0,Y 587.305,Z 230.327,A -85,B 0,C 180,E1 -1304.111,E2 -1304.111} C_VEL
LIN {X 0,Y 587.279,Z 230.328,A -85,B 0,C 180,E1 -1306.99,E2 -1306.99} C_VEL
LIN {X 0,Y 587.308,Z 230.331,A -85,B 0,C 180,E1 -1309.745,E2 -1309.745} C_VEL
LIN {X 0,Y 587.346,Z 230.319,A -85,B 0,C 180,E1 -1312.392,E2 -1312.392} C_VEL
LIN {X 0,Y 587.261,Z 230.333,A -85,B 0,C 180,E1 -1314.468,E2 -1314.468} C_VEL
LIN {X 0,Y 587.344,Z 231.955,A -85,B 0,C 180,E1 -1315.653,E2 -1315.653} C_VEL
LIN {X 0,Y 587.3,Z 236.27,A -85,B 0,C 180,E1 -1318.229,E2 -1318.229} C_VEL
LIN {X 0,Y 587.277,Z 240.795,A -85,B 0,C 180,E1 -1320.88,E2 -1320.88} C_VEL
LIN {X 0,Y 587.217,Z 245.751,A -85,B 0,C 180,E1 -1323.716,E2 -1323.716} C_VEL
LIN {X 0,Y 587.21,Z 249.804,A -85,B 0,C 180,E1 -1325.988,E2 -1325.988} C_VEL
LIN {X 0,Y 587.177,Z 253.951,A -85,B 0,C 180,E1 -1328.22,E2 -1328.22} C_VEL
LIN {X 0,Y 587.203,Z 259.481,A -85,B 0,C 180,E1 -1331.146,E2 -1331.146} C_VEL
LIN {X 0,Y 587.168,Z 265.011,A -85,B 0,C 180,E1 -1334.02,E2 -1334.02} C_VEL
LIN {X 0,Y 587.168,Z 270.54,A -85,B 0,C 180,E1 -1336.855,E2 -1336.855} C_VEL
LIN {X 0,Y 587.158,Z 272.528,A -85,B 0,C 180,E1 -1337.865,E2 -1337.865} C_VEL
LIN {X 0,Y 587.722,Z 277.446,A -85,B 0,C 180,E1 -1337.986,E2 -1337.986} C_VEL
LIN {X 0,Y 587.664,Z 289.891,A -85,B 0,C 180,E1 -1338.315,E2 -1338.315} C_VEL
LIN {X 0,Y 587.59,Z 302.858,A -85,B 0,C 180,E1 -1338.81,E2 -1338.81} C_VEL
LIN {X 0,Y 587.499,Z 314.538,A -85,B 0,C 180,E1 -1339.402,E2 -1339.402} C_VEL
LIN {X 0,Y 587.429,Z 325.322,A -85,B 0,C 180,E1 -1340.097,E2 -1340.097} C_VEL
LIN {X 0,Y 587.357,Z 335.098,A -85,B 0,C 180,E1 -1340.878,E2 -1340.878} C_VEL
LIN {X 0,Y 587.302,Z 343.991,A -85,B 0,C 180,E1 -1341.744,E2 -1341.744} C_VEL
LIN {X 0,Y 587.274,Z 352.676,A -85,B 0,C 180,E1 -1342.781,E2 -1342.781} C_VEL
LIN {X 0,Y 587.214,Z 359.604,A -85,B 0,C 180,E1 -1343.816,E2 -1343.816} C_VEL
LIN {X 0,Y 587.167,Z 365.154,A -85,B 0,C 180,E1 -1344.85,E2 -1344.85} C_VEL
LIN {X 0,Y 587.182,Z 369.516,A -85,B 0,C 180,E1 -1345.882,E2 -1345.882} C_VEL
LIN {X 0,Y 587.194,Z 371.819,A -85,B 0,C 180,E1 -1346.569,E2 -1346.569} C_VEL
LIN {X 0,Y 587.131,Z 373.697,A -85,B 0,C 180,E1 -1347.256,E2 -1347.256} C_VEL
LIN {X 0,Y 587.139,Z 375.127,A -85,B 0,C 180,E1 -1347.942,E2 -1347.942} C_VEL
LIN {X 0,Y 587.14,Z 376.754,A -85,B 0,C 180,E1 -1349.314,E2 -1349.314} C_VEL
LIN {X 0,Y 587.137,Z 376.996,A -85,B 0,C 180,E1 -1350,E2 -1350} C_VEL
LIN {X 0,Y 587.14,Z 376.815,A -85,B 0,C 180,E1 -1350.686,E2 -1350.686} C_VEL
LIN {X 0,Y 587.138,Z 375.274,A -85,B 0,C 180,E1 -1352.058,E2 -1352.058} C_VEL
LIN {X 0,Y 587.133,Z 373.913,A -85,B 0,C 180,E1 -1352.744,E2 -1352.744} C_VEL
LIN {X 0,Y 587.213,Z 371.036,A -85,B 0,C 180,E1 -1353.774,E2 -1353.774} C_VEL
LIN {X 0,Y 587.147,Z 367.136,A -85,B 0,C 180,E1 -1354.806,E2 -1354.806} C_VEL
LIN {X 0,Y 587.229,Z 362.104,A -85,B 0,C 180,E1 -1355.839,E2 -1355.839} C_VEL
LIN {X 0,Y 587.23,Z 355.783,A -85,B 0,C 180,E1 -1356.874,E2 -1356.874} C_VEL
LIN {X 0,Y 587.288,Z 347.864,A -85,B 0,C 180,E1 -1357.91,E2 -1357.91} C_VEL
LIN {X 0,Y 587.343,Z 338.016,A -85,B 0,C 180,E1 -1358.949,E2 -1358.949} C_VEL
LIN {X 0,Y 587.411,Z 327.695,A -85,B 0,C 180,E1 -1359.817,E2 -1359.817} C_VEL
LIN {X 0,Y 587.496,Z 316.065,A -85,B 0,C 180,E1 -1360.599,E2 -1360.599} C_VEL
LIN {X 0,Y 587.591,Z 305.113,A -85,B 0,C 180,E1 -1361.179,E2 -1361.179} C_VEL
LIN {X 0,Y 587.615,Z 292.44,A -85,B 0,C 180,E1 -1361.69,E2 -1361.69} C_VEL
LIN {X 0,Y 587.714,Z 279.484,A -85,B 0,C 180,E1 -1362.058,E2 -1362.058} C_VEL
LIN {X 0,Y 587.4,Z 274.142,A -85,B 0,C 180,E1 -1362.174,E2 -1362.174} C_VEL
LIN {X 0,Y 587.16,Z 272.532,A -85,B 0,C 180,E1 -1362.223,E2 -1362.223} C_VEL
LIN {X 0,Y 587.182,Z 267.951,A -85,B 0,C 180,E1 -1364.558,E2 -1364.558} C_VEL
LIN {X 0,Y 587.183,Z 262.419,A -85,B 0,C 180,E1 -1367.411,E2 -1367.411} C_VEL
LIN {X 0,Y 587.187,Z 258.269,A -85,B 0,C 180,E1 -1369.581,E2 -1369.581} C_VEL
LIN {X 0,Y 587.178,Z 254.12,A -85,B 0,C 180,E1 -1371.78,E2 -1371.78} C_VEL
LIN {X 0,Y 587.204,Z 248.986,A -85,B 0,C 180,E1 -1374.548,E2 -1374.548} C_VEL
LIN {X 0,Y 587.231,Z 244.567,A -85,B 0,C 180,E1 -1377.051,E2 -1377.051} C_VEL
LIN {X 0,Y 587.25,Z 240.52,A -85,B 0,C 180,E1 -1379.385,E2 -1379.385} C_VEL
LIN {X 0,Y 587.28,Z 235.055,A -85,B 0,C 180,E1 -1382.583,E2 -1382.583} C_VEL
LIN {X 0,Y 587.292,Z 230.933,A -85,B 0,C 180,E1 -1385.058,E2 -1385.058} C_VEL
LIN {X 0,Y 587.265,Z 230.334,A -85,B 0,C 180,E1 -1385.533,E2 -1385.533} C_VEL
LIN {X 0,Y 587.343,Z 230.32,A -85,B 0,C 180,E1 -1387.839,E2 -1387.839} C_VEL
LIN {X 0,Y 587.311,Z 230.329,A -85,B 0,C 180,E1 -1390.255,E2 -1390.255} C_VEL
LIN {X 0,Y 587.286,Z 230.327,A -85,B 0,C 180,E1 -1393.115,E2 -1393.115} C_VEL
LIN {X 0,Y 587.301,Z 230.327,A -85,B 0,C 180,E1 -1396.047,E2 -1396.047} C_VEL
LIN {X 0,Y 587.337,Z 230.328,A -85,B 0,C 180,E1 -1398.925,E2 -1398.925} C_VEL
LIN {X 0,Y 587.326,Z 230.322,A -85,B 0,C 180,E1 -1401.52,E2 -1401.52} C_VEL
LIN {X 0,Y 587.3,Z 230.333,A -85,B 0,C 180,E1 -1404.1,E2 -1404.1} C_VEL
LIN {X 0,Y 587.337,Z 230.321,A -85,B 0,C 180,E1 -1406.889,E2 -1406.889} C_VEL
LIN {X 0,Y 587.307,Z 230.328,A -85,B 0,C 180,E1 -1409.496,E2 -1409.496} C_VEL
LIN {X 0,Y 587.345,Z 230.323,A -85,B 0,C 180,E1 -1412.309,E2 -1412.309} C_VEL
LIN {X 0,Y 587.339,Z 230.327,A -85,B 0,C 180,E1 -1414.483,E2 -1414.483} C_VEL
LIN {X 0,Y 587.342,Z 230.323,A -85,B 0,C 180,E1 -1417.486,E2 -1417.486} C_VEL
LIN {X 0,Y 587.327,Z 230.327,A -85,B 0,C 180,E1 -1419.695,E2 -1419.695} C_VEL
LIN {X 0,Y 587.284,Z 230.328,A -85,B 0,C 180,E1 -1421.872,E2 -1421.872} C_VEL
LIN {X 0,Y 587.312,Z 230.33,A -85,B 0,C 180,E1 -1424.736,E2 -1424.736} C_VEL
LIN {X 0,Y 587.31,Z 230.326,A -85,B 0,C 180,E1 -1426.858,E2 -1426.858} C_VEL
LIN {X 0,Y 587.34,Z 230.327,A -85,B 0,C 180,E1 -1429.66,E2 -1429.66} C_VEL
LIN {X 0,Y 587.36,Z 230.318,A -85,B 0,C 180,E1 -1432.437,E2 -1432.437} C_VEL
LIN {X 0,Y 587.341,Z 230.324,A -85,B 0,C 180,E1 -1435.195,E2 -1435.195} C_VEL
LIN {X 0,Y 587.346,Z 230.322,A -85,B 0,C 180,E1 -1437.943,E2 -1437.943} C_VEL
LIN {X 0,Y 587.388,Z 230.315,A -85,B 0,C 180,E1 -1440.686,E2 -1440.686} C_VEL
LIN {X 0,Y 587.332,Z 230.329,A -85,B 0,C 180,E1 -1443.43,E2 -1443.43} C_VEL
LIN {X 0,Y 587.357,Z 230.322,A -85,B 0,C 180,E1 -1445.493,E2 -1445.493} C_VEL
LIN {X 0,Y 587.343,Z 230.32,A -85,B 0,C 180,E1 -1447.563,E2 -1447.563} C_VEL
LIN {X 0,Y 587.292,Z 230.334,A -85,B 0,C 180,E1 -1450.341,E2 -1450.341} C_VEL
LIN {X 0,Y 587.325,Z 230.325,A -85,B 0,C 180,E1 -1452.438,E2 -1452.438} C_VEL
LIN {X 0,Y 587.335,Z 230.321,A -85,B 0,C 180,E1 -1454.554,E2 -1454.554} C_VEL
LIN {X 0,Y 587.348,Z 230.324,A -85,B 0,C 180,E1 -1457.406,E2 -1457.406} C_VEL
LIN {X 0,Y 587.331,Z 230.325,A -85,B 0,C 180,E1 -1460.305,E2 -1460.305} C_VEL
LIN {X 0,Y 587.309,Z 230.324,A -85,B 0,C 180,E1 -1463.259,E2 -1463.259} C_VEL
LIN {X 0,Y 587.309,Z 230.326,A -85,B 0,C 180,E1 -1466.17,E2 -1466.17} C_VEL
LIN {X 0,Y 587.345,Z 230.327,A -85,B 0,C 180,E1 -1469.132,E2 -1469.132} C_VEL
LIN {X 0,Y 587.352,Z 230.319,A -85,B 0,C 180,E1 -1471.836,E2 -1471.836} C_VEL
LIN {X 0,Y 587.347,Z 230.326,A -85,B 0,C 180,E1 -1474.347,E2 -1474.347} C_VEL
LIN {X 0,Y 587.335,Z 230.327,A -85,B 0,C 180,E1 -1477.609,E2 -1477.609} C_VEL
LIN {X 0,Y 587.293,Z 230.326,A -85,B 0,C 180,E1 -1480.256,E2 -1480.256} C_VEL
LIN {X 0,Y 587.307,Z 230.329,A -85,B 0,C 180,E1 -1483.117,E2 -1483.117} C_VEL
LIN {X 0,Y 587.315,Z 230.328,A -85,B 0,C 180,E1 -1486.048,E2 -1486.048} C_VEL
LIN {X 0,Y 587.337,Z 230.321,A -85,B 0,C 180,E1 -1488.925,E2 -1488.925} C_VEL
LIN {X 0,Y 587.318,Z 230.33,A -85,B 0,C 180,E1 -1491.519,E2 -1491.519} C_VEL
LIN {X 0,Y 587.333,Z 230.519,A -85,B 0,C 180,E1 -1494.103,E2 -1494.103} C_VEL
LIN {X 0,Y 587.486,Z 234.52,A -85,B 0,C 180,E1 -1495.633,E2 -1495.633} C_VEL
LIN {X 0,Y 587.455,Z 241.589,A -85,B 0,C 180,E1 -1498.238,E2 -1498.238} C_VEL
LIN {X 0,Y 587.396,Z 249.043,A -85,B 0,C 180,E1 -1500.859,E2 -1500.859} C_VEL
LIN {X 0,Y 587.366,Z 257.661,A -85,B 0,C 180,E1 -1503.818,E2 -1503.818} C_VEL
LIN {X 0,Y 587.331,Z 266.334,A -85,B 0,C 180,E1 -1506.741,E2 -1506.741} C_VEL
LIN {X 0,Y 587.295,Z 274.141,A -85,B 0,C 180,E1 -1509.333,E2 -1509.333} C_VEL
LIN {X 0,Y 587.281,Z 283.03,A -85,B 0,C 180,E1 -1512.232,E2 -1512.232} C_VEL
LIN {X 0,Y 587.219,Z 291.935,A -85,B 0,C 180,E1 -1515.089,E2 -1515.089} C_VEL
LIN {X 0,Y 587.173,Z 300.491,A -85,B 0,C 180,E1 -1517.799,E2 -1517.799} C_VEL
LIN {X 0,Y 587.747,Z 305.224,A -85,B 0,C 180,E1 -1517.899,E2 -1517.899} C_VEL
LIN {X 0,Y 587.68,Z 318.493,A -85,B 0,C 180,E1 -1518.226,E2 -1518.226} C_VEL
LIN {X 0,Y 587.566,Z 330.458,A -85,B 0,C 180,E1 -1518.658,E2 -1518.658} C_VEL
LIN {X 0,Y 587.49,Z 342.209,A -85,B 0,C 180,E1 -1519.227,E2 -1519.227} C_VEL
LIN {X 0,Y 587.457,Z 353.477,A -85,B 0,C 180,E1 -1519.923,E2 -1519.923} C_VEL
LIN {X 0,Y 587.384,Z 363.646,A -85,B 0,C 180,E1 -1520.704,E2 -1520.704} C_VEL
LIN {X 0,Y 587.34,Z 372.786,A -85,B 0,C 180,E1 -1521.571,E2 -1521.571} C_VEL
LIN {X 0,Y 587.259,Z 381.69,A -85,B 0,C 180,E1 -1522.608,E2 -1522.608} C_VEL
LIN {X 0,Y 587.195,Z 388.745,A -85,B 0,C 180,E1 -1523.627,E2 -1523.627} C_VEL
LIN {X 0,Y 587.211,Z 393.68,A -85,B 0,C 180,E1 -1524.506,E2 -1524.506} C_VEL
LIN {X 0,Y 587.188,Z 398.371,A -85,B 0,C 180,E1 -1525.538,E2 -1525.538} C_VEL
LIN {X 0,Y 587.193,Z 401.956,A -85,B 0,C 180,E1 -1526.569,E2 -1526.569} C_VEL
LIN {X 0,Y 587.132,Z 403.808,A -85,B 0,C 180,E1 -1527.256,E2 -1527.256} C_VEL
LIN {X 0,Y 587.141,Z 405.2,A -85,B 0,C 180,E1 -1527.942,E2 -1527.942} C_VEL
LIN {X 0,Y 587.14,Z 406.784,A -85,B 0,C 180,E1 -1529.314,E2 -1529.314} C_VEL
LIN {X 0,Y 587.137,Z 407,A -85,B 0,C 180,E1 -1530,E2 -1530} C_VEL
LIN {X 0,Y 587.147,Z 406.185,A -85,B 0,C 180,E1 -1531.372,E2 -1531.372} C_VEL
LIN {X 0,Y 587.141,Z 405.201,A -85,B 0,C 180,E1 -1532.058,E2 -1532.058} C_VEL
LIN {X 0,Y 587.132,Z 403.81,A -85,B 0,C 180,E1 -1532.744,E2 -1532.744} C_VEL
LIN {X 0,Y 587.213,Z 400.896,A -85,B 0,C 180,E1 -1533.774,E2 -1533.774} C_VEL
LIN {X 0,Y 587.147,Z 396.95,A -85,B 0,C 180,E1 -1534.806,E2 -1534.806} C_VEL
LIN {X 0,Y 587.218,Z 390.878,A -85,B 0,C 180,E1 -1536.011,E2 -1536.011} C_VEL
LIN {X 0,Y 587.245,Z 384.237,A -85,B 0,C 180,E1 -1537.046,E2 -1537.046} C_VEL
LIN {X 0,Y 587.299,Z 375.99,A -85,B 0,C 180,E1 -1538.083,E2 -1538.083} C_VEL
LIN {X 0,Y 587.343,Z 367.538,A -85,B 0,C 180,E1 -1538.949,E2 -1538.949} C_VEL
LIN {X 0,Y 587.415,Z 357.096,A -85,B 0,C 180,E1 -1539.816,E2 -1539.816} C_VEL
LIN {X 0,Y 587.451,Z 346.758,A -85,B 0,C 180,E1 -1540.512,E2 -1540.512} C_VEL
LIN {X 0,Y 587.529,Z 335.169,A -85,B 0,C 180,E1 -1541.133,E2 -1541.133} C_VEL
LIN {X 0,Y 587.607,Z 322.698,A -85,B 0,C 180,E1 -1541.636,E2 -1541.636} C_VEL
LIN {X 0,Y 587.744,Z 309.436,A -85,B 0,C 180,E1 -1542.013,E2 -1542.013} C_VEL
LIN {X 0,Y 587.528,Z 302.65,A -85,B 0,C 180,E1 -1542.155,E2 -1542.155} C_VEL
LIN {X 0,Y 587.173,Z 300.492,A -85,B 0,C 180,E1 -1542.2,E2 -1542.2} C_VEL
LIN {X 0,Y 587.219,Z 291.935,A -85,B 0,C 180,E1 -1544.911,E2 -1544.911} C_VEL
LIN {X 0,Y 587.281,Z 283.031,A -85,B 0,C 180,E1 -1547.768,E2 -1547.768} C_VEL
LIN {X 0,Y 587.295,Z 274.142,A -85,B 0,C 180,E1 -1550.667,E2 -1550.667} C_VEL
LIN {X 0,Y 587.346,Z 265.222,A -85,B 0,C 180,E1 -1553.631,E2 -1553.631} C_VEL
LIN {X 0,Y 587.365,Z 257.38,A -85,B 0,C 180,E1 -1556.277,E2 -1556.277} C_VEL
LIN {X 0,Y 587.421,Z 248.366,A -85,B 0,C 180,E1 -1559.376,E2 -1559.376} C_VEL
LIN {X 0,Y 587.478,Z 240.435,A -85,B 0,C 180,E1 -1562.174,E2 -1562.174} C_VEL
LIN {X 0,Y 587.531,Z 232.724,A -85,B 0,C 180,E1 -1565.042,E2 -1565.042} C_VEL
LIN {X 0,Y 587.302,Z 230.331,A -85,B 0,C 180,E1 -1566.005,E2 -1566.005} C_VEL
LIN {X 0,Y 587.317,Z 230.33,A -85,B 0,C 180,E1 -1568.48,E2 -1568.48} C_VEL
LIN {X 0,Y 587.336,Z 230.322,A -85,B 0,C 180,E1 -1571.157,E2 -1571.157} C_VEL
LIN {X 0,Y 587.314,Z 230.326,A -85,B 0,C 180,E1 -1574.112,E2 -1574.112} C_VEL
LIN {X 0,Y 587.302,Z 230.331,A -85,B 0,C 180,E1 -1576.992,E2 -1576.992} C_VEL
LIN {X 0,Y 587.292,Z 230.326,A -85,B 0,C 180,E1 -1579.744,E2 -1579.744} C_VEL
LIN {X 0,Y 587.334,Z 230.327,A -85,B 0,C 180,E1 -1582.391,E2 -1582.391} C_VEL
LIN {X 0,Y 587.346,Z 230.326,A -85,B 0,C 180,E1 -1585.653,E2 -1585.653} C_VEL
LIN {X 0,Y 587.355,Z 230.319,A -85,B 0,C 180,E1 -1588.232,E2 -1588.232} C_VEL
LIN {X 0,Y 587.345,Z 230.327,A -85,B 0,C 180,E1 -1590.868,E2 -1590.868} C_VEL
LIN {X 0,Y 587.309,Z 230.326,A -85,B 0,C 180,E1 -1593.829,E2 -1593.829} C_VEL
LIN {X 0,Y 587.307,Z 230.324,A -85,B 0,C 180,E1 -1596.741,E2 -1596.741} C_VEL
LIN {X 0,Y 587.33,Z 230.326,A -85,B 0,C 180,E1 -1599.695,E2 -1599.695} C_VEL
LIN {X 0,Y 587.347,Z 230.324,A -85,B 0,C 180,E1 -1602.594,E2 -1602.594} C_VEL
LIN {X 0,Y 587.342,Z 230.321,A -85,B 0,C 180,E1 -1605.75,E2 -1605.75} C_VEL
LIN {X 0,Y 587.321,Z 230.326,A -85,B 0,C 180,E1 -1608.263,E2 -1608.263} C_VEL
LIN {X 0,Y 587.316,Z 230.325,A -85,B 0,C 180,E1 -1611.051,E2 -1611.051} C_VEL
LIN {X 0,Y 587.315,Z 230.324,A -85,B 0,C 180,E1 -1613.817,E2 -1613.817} C_VEL
LIN {X 0,Y 587.312,Z 230.324,A -85,B 0,C 180,E1 -1615.883,E2 -1615.883} C_VEL
LIN {X 0,Y 587.37,Z 230.32,A -85,B 0,C 180,E1 -1617.943,E2 -1617.943} C_VEL
LIN {X 0,Y 587.372,Z 230.317,A -85,B 0,C 180,E1 -1620.686,E2 -1620.686} C_VEL
LIN {X 0,Y 587.316,Z 230.331,A -85,B 0,C 180,E1 -1623.43,E2 -1623.43} C_VEL
LIN {X 0,Y 587.353,Z 230.321,A -85,B 0,C 180,E1 -1625.493,E2 -1625.493} C_VEL
LIN {X 0,Y 587.334,Z 230.324,A -85,B 0,C 180,E1 -1628.256,E2 -1628.256} C_VEL
LIN {X 0,Y 587.352,Z 230.319,A -85,B 0,C 180,E1 -1631.134,E2 -1631.134} C_VEL
LIN {X 0,Y 587.353,Z 230.325,A -85,B 0,C 180,E1 -1633.846,E2 -1633.846} C_VEL
LIN {X 0,Y 587.328,Z 230.325,A -85,B 0,C 180,E1 -1636.807,E2 -1636.807} C_VEL
LIN {X 0,Y 587.286,Z 230.328,A -85,B 0,C 180,E1 -1638.293,E2 -1638.293} C_VEL
LIN {X 0,Y 586.653,Z 230.413,A -85,B 0,C 180,E1 -1638.865,E2 -1638.865} C_VEL
LIN {X 0,Y 583.842,Z 230.76,A -85,B 0,C 180,E1 -1639.794,E2 -1639.794} C_VEL
LIN {X 0,Y 581.436,Z 231.063,A -85,B 0,C 180,E1 -1640.541,E2 -1640.541} C_VEL
LIN {X 0,Y 580.382,Z 231.188,A -85,B 0,C 180,E1 -1641.118,E2 -1641.118} C_VEL
LIN {X 0,Y 580.286,Z 231.199,A -85,B 0,C 180,E1 -1641.313,E2 -1641.313} C_VEL
LIN {X 0,Y 580.301,Z 231.2,A -85,B 0,C 180,E1 -1644.316,E2 -1644.316} C_VEL
LIN {X 0,Y 580.281,Z 231.2,A -85,B 0,C 180,E1 -1646.623,E2 -1646.623} C_VEL
LIN {X 0,Y 580.276,Z 231.206,A -85,B 0,C 180,E1 -1649.305,E2 -1649.305} C_VEL
LIN {X 0,Y 580.296,Z 231.201,A -85,B 0,C 180,E1 -1652.201,E2 -1652.201} C_VEL
LIN {X 0,Y 580.28,Z 231.201,A -85,B 0,C 180,E1 -1654.697,E2 -1654.697} C_VEL
LIN {X 0,Y 580.29,Z 231.2,A -85,B 0,C 180,E1 -1657.269,E2 -1657.269} C_VEL
LIN {X 0,Y 580.293,Z 231.198,A -85,B 0,C 180,E1 -1660.27,E2 -1660.27} C_VEL
LIN {X 0,Y 580.276,Z 231.206,A -85,B 0,C 180,E1 -1662.707,E2 -1662.707} C_VEL
LIN {X 0,Y 580.238,Z 231.206,A -85,B 0,C 180,E1 -1665.613,E2 -1665.613} C_VEL
LIN {X 0,Y 580.247,Z 231.208,A -85,B 0,C 180,E1 -1668.228,E2 -1668.228} C_VEL
LIN {X 0,Y 580.276,Z 231.202,A -85,B 0,C 180,E1 -1670.965,E2 -1670.965} C_VEL
LIN {X 0,Y 580.265,Z 231.204,A -85,B 0,C 180,E1 -1673.596,E2 -1673.596} C_VEL
LIN {X 0,Y 580.219,Z 231.21,A -85,B 0,C 180,E1 -1674.45,E2 -1674.45} C_VEL
LIN {X 0,Y 580.29,Z 232.468,A -85,B 0,C 180,E1 -1675.443,E2 -1675.443} C_VEL
LIN {X 0,Y 580.238,Z 236.676,A -85,B 0,C 180,E1 -1677.98,E2 -1677.98} C_VEL
LIN {X 0,Y 580.225,Z 241.775,A -85,B 0,C 180,E1 -1681.02,E2 -1681.02} C_VEL
LIN {X 0,Y 580.151,Z 246.415,A -85,B 0,C 180,E1 -1683.695,E2 -1683.695} C_VEL
LIN {X 0,Y 580.133,Z 251.223,A -85,B 0,C 180,E1 -1686.436,E2 -1686.436} C_VEL
LIN {X 0,Y 580.114,Z 256.717,A -85,B 0,C 180,E1 -1689.431,E2 -1689.431} C_VEL
LIN {X 0,Y 580.093,Z 260.864,A -85,B 0,C 180,E1 -1691.639,E2 -1691.639} C_VEL
LIN {X 0,Y 580.094,Z 265.012,A -85,B 0,C 180,E1 -1693.82,E2 -1693.82} C_VEL
LIN {X 0,Y 580.093,Z 269.159,A -85,B 0,C 180,E1 -1695.977,E2 -1695.977} C_VEL
LIN {X 0,Y 580.078,Z 272.529,A -85,B 0,C 180,E1 -1697.715,E2 -1697.715} C_VEL
LIN {X 0,Y 580.793,Z 278.492,A -85,B 0,C 180,E1 -1697.863,E2 -1697.863} C_VEL
LIN {X 0,Y 580.706,Z 291.154,A -85,B 0,C 180,E1 -1698.216,E2 -1698.216} C_VEL
LIN {X 0,Y 580.619,Z 303.267,A -85,B 0,C 180,E1 -1698.691,E2 -1698.691} C_VEL
LIN {X 0,Y 580.52,Z 314.55,A -85,B 0,C 180,E1 -1699.273,E2 -1699.273} C_VEL
LIN {X 0,Y 580.431,Z 325.327,A -85,B 0,C 180,E1 -1699.976,E2 -1699.976} C_VEL
LIN {X 0,Y 580.333,Z 335.103,A -85,B 0,C 180,E1 -1700.766,E2 -1700.766} C_VEL
LIN {X 0,Y 580.264,Z 343.996,A -85,B 0,C 180,E1 -1701.643,E2 -1701.643} C_VEL
LIN {X 0,Y 580.206,Z 352.68,A -85,B 0,C 180,E1 -1702.693,E2 -1702.693} C_VEL
LIN {X 0,Y 580.137,Z 359.608,A -85,B 0,C 180,E1 -1703.741,E2 -1703.741} C_VEL
LIN {X 0,Y 580.086,Z 365.157,A -85,B 0,C 180,E1 -1704.787,E2 -1704.787} C_VEL
LIN {X 0,Y 580.105,Z 369.518,A -85,B 0,C 180,E1 -1705.832,E2 -1705.832} C_VEL
LIN {X 0,Y 580.123,Z 371.822,A -85,B 0,C 180,E1 -1706.527,E2 -1706.527} C_VEL
LIN {X 0,Y 580.043,Z 373.699,A -85,B 0,C 180,E1 -1707.222,E2 -1707.222} C_VEL
LIN {X 0,Y 580.038,Z 375.127,A -85,B 0,C 180,E1 -1707.917,E2 -1707.917} C_VEL
LIN {X 0,Y 580.04,Z 376.755,A -85,B 0,C 180,E1 -1709.306,E2 -1709.306} C_VEL
LIN {X 0,Y 580.038,Z 376.996,A -85,B 0,C 180,E1 -1710,E2 -1710} C_VEL
LIN {X 0,Y 580.04,Z 376.815,A -85,B 0,C 180,E1 -1710.694,E2 -1710.694} C_VEL
LIN {X 0,Y 580.037,Z 375.272,A -85,B 0,C 180,E1 -1712.083,E2 -1712.083} C_VEL
LIN {X 0,Y 580.044,Z 373.911,A -85,B 0,C 180,E1 -1712.778,E2 -1712.778} C_VEL
LIN {X 0,Y 580.109,Z 371.034,A -85,B 0,C 180,E1 -1713.821,E2 -1713.821} C_VEL
LIN {X 0,Y 580.053,Z 367.133,A -85,B 0,C 180,E1 -1714.865,E2 -1714.865} C_VEL
LIN {X 0,Y 580.162,Z 362.101,A -85,B 0,C 180,E1 -1715.91,E2 -1715.91} C_VEL
LIN {X 0,Y 580.158,Z 355.779,A -85,B 0,C 180,E1 -1716.958,E2 -1716.958} C_VEL
LIN {X 0,Y 580.241,Z 347.859,A -85,B 0,C 180,E1 -1718.007,E2 -1718.007} C_VEL
LIN {X 0,Y 580.308,Z 338.01,A -85,B 0,C 180,E1 -1719.058,E2 -1719.058} C_VEL
LIN {X 0,Y 580.404,Z 327.69,A -85,B 0,C 180,E1 -1719.936,E2 -1719.936} C_VEL
LIN {X 0,Y 580.492,Z 316.054,A -85,B 0,C 180,E1 -1720.728,E2 -1720.728} C_VEL
LIN {X 0,Y 580.631,Z 304.283,A -85,B 0,C 180,E1 -1721.353,E2 -1721.353} C_VEL
LIN {X 0,Y 580.679,Z 292.621,A -85,B 0,C 180,E1 -1721.825,E2 -1721.825} C_VEL
LIN {X 0,Y 580.78,Z 279.46,A -85,B 0,C 180,E1 -1722.204,E2 -1722.204} C_VEL
LIN {X 0,Y 580.478,Z 275.254,A -85,B 0,C 180,E1 -1722.299,E2 -1722.299} C_VEL
LIN {X 0,Y 580.095,Z 272.531,A -85,B 0,C 180,E1 -1722.374,E2 -1722.374} C_VEL
LIN {X 0,Y 580.106,Z 267.95,A -85,B 0,C 180,E1 -1724.739,E2 -1724.739} C_VEL
LIN {X 0,Y 580.079,Z 262.417,A -85,B 0,C 180,E1 -1727.631,E2 -1727.631} C_VEL
LIN {X 0,Y 580.099,Z 258.268,A -85,B 0,C 180,E1 -1729.83,E2 -1729.83} C_VEL
LIN {X 0,Y 580.12,Z 254.118,A -85,B 0,C 180,E1 -1732.059,E2 -1732.059} C_VEL
LIN {X 0,Y 580.151,Z 249.39,A -85,B 0,C 180,E1 -1734.693,E2 -1734.693} C_VEL
LIN {X 0,Y 580.217,Z 243.919,A -85,B 0,C 180,E1 -1737.843,E2 -1737.843} C_VEL
LIN {X 0,Y 580.186,Z 239.074,A -85,B 0,C 180,E1 -1740.678,E2 -1740.678} C_VEL
LIN {X 0,Y 580.231,Z 234.691,A -85,B 0,C 180,E1 -1743.305,E2 -1743.305} C_VEL
LIN {X 0,Y 580.27,Z 232.387,A -85,B 0,C 180,E1 -1744.698,E2 -1744.698} C_VEL
LIN {X 0,Y 580.222,Z 231.211,A -85,B 0,C 180,E1 -1745.55,E2 -1745.55} C_VEL
LIN {X 0,Y 580.291,Z 231.199,A -85,B 0,C 180,E1 -1748.146,E2 -1748.146} C_VEL
LIN {X 0,Y 580.295,Z 231.2,A -85,B 0,C 180,E1 -1750.844,E2 -1750.844} C_VEL
LIN {X 0,Y 580.229,Z 231.212,A -85,B 0,C 180,E1 -1753.663,E2 -1753.663} C_VEL
LIN {X 0,Y 580.246,Z 231.205,A -85,B 0,C 180,E1 -1756.613,E2 -1756.613} C_VEL
LIN {X 0,Y 580.3,Z 231.202,A -85,B 0,C 180,E1 -1759.156,E2 -1759.156} C_VEL
LIN {X 0,Y 580.291,Z 231.2,A -85,B 0,C 180,E1 -1761.927,E2 -1761.927} C_VEL
LIN {X 0,Y 580.255,Z 231.205,A -85,B 0,C 180,E1 -1764.453,E2 -1764.453} C_VEL
LIN {X 0,Y 580.289,Z 231.2,A -85,B 0,C 180,E1 -1766.975,E2 -1766.975} C_VEL
LIN {X 0,Y 580.271,Z 231.206,A -85,B 0,C 180,E1 -1769.423,E2 -1769.423} C_VEL
LIN {X 0,Y 580.293,Z 231.2,A -85,B 0,C 180,E1 -1772.143,E2 -1772.143} C_VEL
LIN {X 0,Y 580.311,Z 231.197,A -85,B 0,C 180,E1 -1774.92,E2 -1774.92} C_VEL
LIN {X 0,Y 580.273,Z 231.206,A -85,B 0,C 180,E1 -1777.947,E2 -1777.947} C_VEL
LIN {X 0,Y 580.295,Z 231.201,A -85,B 0,C 180,E1 -1780.913,E2 -1780.913} C_VEL
LIN {X 0,Y 580.253,Z 231.203,A -85,B 0,C 180,E1 -1783.825,E2 -1783.825} C_VEL
LIN {X 0,Y 580.267,Z 231.205,A -85,B 0,C 180,E1 -1786.696,E2 -1786.696} C_VEL
LIN {X 0,Y 580.31,Z 231.196,A -85,B 0,C 180,E1 -1788.827,E2 -1788.827} C_VEL
LIN {X 0,Y 580.304,Z 231.202,A -85,B 0,C 180,E1 -1791.644,E2 -1791.644} C_VEL
LIN {X 0,Y 580.318,Z 231.196,A -85,B 0,C 180,E1 -1794.44,E2 -1794.44} C_VEL
LIN {X 0,Y 580.312,Z 231.197,A -85,B 0,C 180,E1 -1797.223,E2 -1797.223} C_VEL
LIN {X 0,Y 580.351,Z 231.198,A -85,B 0,C 180,E1 -1800,E2 -1800} C_VEL
LIN {X 0,Y 580.342,Z 231.193,A -85,B 0,C 180,E1 -1802.776,E2 -1802.776} C_VEL
LIN {X 0,Y 580.323,Z 231.197,A -85,B 0,C 180,E1 -1805.56,E2 -1805.56} C_VEL
LIN {X 0,Y 580.291,Z 231.198,A -85,B 0,C 180,E1 -1807.656,E2 -1807.656} C_VEL
LIN {X 0,Y 580.254,Z 231.209,A -85,B 0,C 180,E1 -1810.468,E2 -1810.468} C_VEL
LIN {X 0,Y 580.292,Z 231.199,A -85,B 0,C 180,E1 -1812.592,E2 -1812.592} C_VEL
LIN {X 0,Y 580.283,Z 231.2,A -85,B 0,C 180,E1 -1814.734,E2 -1814.734} C_VEL
LIN {X 0,Y 580.295,Z 231.2,A -85,B 0,C 180,E1 -1817.625,E2 -1817.625} C_VEL
LIN {X 0,Y 580.291,Z 231.199,A -85,B 0,C 180,E1 -1819.823,E2 -1819.823} C_VEL
LIN {X 0,Y 580.27,Z 231.205,A -85,B 0,C 180,E1 -1822.053,E2 -1822.053} C_VEL
LIN {X 0,Y 580.277,Z 231.2,A -85,B 0,C 180,E1 -1825.081,E2 -1825.081} C_VEL
LIN {X 0,Y 580.277,Z 231.2,A -85,B 0,C 180,E1 -1828.187,E2 -1828.187} C_VEL
LIN {X 0,Y 580.28,Z 231.205,A -85,B 0,C 180,E1 -1830.693,E2 -1830.693} C_VEL
LIN {X 0,Y 580.307,Z 231.197,A -85,B 0,C 180,E1 -1833.316,E2 -1833.316} C_VEL
LIN {X 0,Y 580.246,Z 231.208,A -85,B 0,C 180,E1 -1835.756,E2 -1835.756} C_VEL
LIN {X 0,Y 580.277,Z 231.202,A -85,B 0,C 180,E1 -1838.147,E2 -1838.147} C_VEL
LIN {X 0,Y 580.29,Z 231.202,A -85,B 0,C 180,E1 -1840.844,E2 -1840.844} C_VEL
LIN {X 0,Y 580.273,Z 231.201,A -85,B 0,C 180,E1 -1843.659,E2 -1843.659} C_VEL
LIN {X 0,Y 580.277,Z 231.204,A -85,B 0,C 180,E1 -1846.61,E2 -1846.61} C_VEL
LIN {X 0,Y 580.299,Z 231.199,A -85,B 0,C 180,E1 -1849.156,E2 -1849.156} C_VEL
LIN {X 0,Y 580.285,Z 231.202,A -85,B 0,C 180,E1 -1851.928,E2 -1851.928} C_VEL
LIN {X 0,Y 580.299,Z 231.361,A -85,B 0,C 180,E1 -1853.943,E2 -1853.943} C_VEL
LIN {X 0,Y 580.514,Z 235.119,A -85,B 0,C 180,E1 -1855.411,E2 -1855.411} C_VEL
LIN {X 0,Y 580.448,Z 241.884,A -85,B 0,C 180,E1 -1857.947,E2 -1857.947} C_VEL
LIN {X 0,Y 580.38,Z 249.539,A -85,B 0,C 180,E1 -1860.677,E2 -1860.677} C_VEL
LIN {X 0,Y 580.31,Z 257.287,A -85,B 0,C 180,E1 -1863.378,E2 -1863.378} C_VEL
LIN {X 0,Y 580.312,Z 265.204,A -85,B 0,C 180,E1 -1866.064,E2 -1866.064} C_VEL
LIN {X 0,Y 580.263,Z 273.465,A -85,B 0,C 180,E1 -1868.845,E2 -1868.845} C_VEL
LIN {X 0,Y 580.2,Z 281.917,A -85,B 0,C 180,E1 -1871.643,E2 -1871.643} C_VEL
LIN {X 0,Y 580.174,Z 290.822,A -85,B 0,C 180,E1 -1874.544,E2 -1874.544} C_VEL
LIN {X 0,Y 580.13,Z 299.726,A -85,B 0,C 180,E1 -1877.405,E2 -1877.405} C_VEL
LIN {X 0,Y 580.105,Z 300.491,A -85,B 0,C 180,E1 -1877.649,E2 -1877.649} C_VEL
LIN {X 0,Y 580.807,Z 306.364,A -85,B 0,C 180,E1 -1877.775,E2 -1877.775} C_VEL
LIN {X 0,Y 580.731,Z 318.494,A -85,B 0,C 180,E1 -1878.083,E2 -1878.083} C_VEL
LIN {X 0,Y 580.616,Z 330.315,A -85,B 0,C 180,E1 -1878.515,E2 -1878.515} C_VEL
LIN {X 0,Y 580.505,Z 342.208,A -85,B 0,C 180,E1 -1879.096,E2 -1879.096} C_VEL
LIN {X 0,Y 580.446,Z 353.479,A -85,B 0,C 180,E1 -1879.8,E2 -1879.8} C_VEL
LIN {X 0,Y 580.352,Z 363.646,A -85,B 0,C 180,E1 -1880.591,E2 -1880.591} C_VEL
LIN {X 0,Y 580.279,Z 372.786,A -85,B 0,C 180,E1 -1881.468,E2 -1881.468} C_VEL
LIN {X 0,Y 580.199,Z 381.689,A -85,B 0,C 180,E1 -1882.518,E2 -1882.518} C_VEL
LIN {X 0,Y 580.12,Z 388.464,A -85,B 0,C 180,E1 -1883.505,E2 -1883.505} C_VEL
LIN {X 0,Y 580.139,Z 393.68,A -85,B 0,C 180,E1 -1884.438,E2 -1884.438} C_VEL
LIN {X 0,Y 580.108,Z 398.371,A -85,B 0,C 180,E1 -1885.483,E2 -1885.483} C_VEL
LIN {X 0,Y 580.123,Z 401.957,A -85,B 0,C 180,E1 -1886.527,E2 -1886.527} C_VEL
LIN {X 0,Y 580.043,Z 403.808,A -85,B 0,C 180,E1 -1887.222,E2 -1887.222} C_VEL
LIN {X 0,Y 580.04,Z 405.199,A -85,B 0,C 180,E1 -1887.917,E2 -1887.917} C_VEL
LIN {X 0,Y 580.04,Z 406.785,A -85,B 0,C 180,E1 -1889.306,E2 -1889.306} C_VEL
LIN {X 0,Y 580.037,Z 407,A -85,B 0,C 180,E1 -1890,E2 -1890} C_VEL
LIN {X 0,Y 580.047,Z 406.186,A -85,B 0,C 180,E1 -1891.388,E2 -1891.388} C_VEL
LIN {X 0,Y 580.04,Z 405.2,A -85,B 0,C 180,E1 -1892.083,E2 -1892.083} C_VEL
LIN {X 0,Y 580.043,Z 403.81,A -85,B 0,C 180,E1 -1892.778,E2 -1892.778} C_VEL
LIN {X 0,Y 580.11,Z 400.896,A -85,B 0,C 180,E1 -1893.821,E2 -1893.821} C_VEL
LIN {X 0,Y 580.053,Z 396.949,A -85,B 0,C 180,E1 -1894.865,E2 -1894.865} C_VEL
LIN {X 0,Y 580.139,Z 390.877,A -85,B 0,C 180,E1 -1896.085,E2 -1896.085} C_VEL
LIN {X 0,Y 580.184,Z 384.238,A -85,B 0,C 180,E1 -1897.132,E2 -1897.132} C_VEL
LIN {X 0,Y 580.25,Z 375.991,A -85,B 0,C 180,E1 -1898.182,E2 -1898.182} C_VEL
LIN {X 0,Y 580.308,Z 367.538,A -85,B 0,C 180,E1 -1899.058,E2 -1899.058} C_VEL
LIN {X 0,Y 580.412,Z 357.097,A -85,B 0,C 180,E1 -1899.936,E2 -1899.936} C_VEL
LIN {X 0,Y 580.454,Z 346.756,A -85,B 0,C 180,E1 -1900.64,E2 -1900.64} C_VEL
LIN {X 0,Y 580.563,Z 335.59,A -85,B 0,C 180,E1 -1901.248,E2 -1901.248} C_VEL
LIN {X 0,Y 580.63,Z 323.768,A -85,B 0,C 180,E1 -1901.742,E2 -1901.742} C_VEL
LIN {X 0,Y 580.778,Z 310.35,A -85,B 0,C 180,E1 -1902.137,E2 -1902.137} C_VEL
LIN {X 0,Y 580.678,Z 304.086,A -85,B 0,C 180,E1 -1902.272,E2 -1902.272} C_VEL
LIN {X 0,Y 580.105,Z 300.492,A -85,B 0,C 180,E1 -1902.351,E2 -1902.351} C_VEL
LIN {X 0,Y 580.156,Z 291.935,A -85,B 0,C 180,E1 -1905.097,E2 -1905.097} C_VEL
LIN {X 0,Y 580.207,Z 283.031,A -85,B 0,C 180,E1 -1907.992,E2 -1907.992} C_VEL
LIN {X 0,Y 580.239,Z 275.239,A -85,B 0,C 180,E1 -1910.564,E2 -1910.564} C_VEL
LIN {X 0,Y 580.269,Z 267.972,A -85,B 0,C 180,E1 -1913.003,E2 -1913.003} C_VEL
LIN {X 0,Y 580.328,Z 260.671,A -85,B 0,C 180,E1 -1915.462,E2 -1915.462} C_VEL
LIN {X 0,Y 580.349,Z 251.666,A -85,B 0,C 180,E1 -1918.577,E2 -1918.577} C_VEL
LIN {X 0,Y 580.42,Z 243.765,A -85,B 0,C 180,E1 -1921.377,E2 -1921.377} C_VEL
LIN {X 0,Y 580.488,Z 237.093,A -85,B 0,C 180,E1 -1923.843,E2 -1923.843} C_VEL
LIN {X 0,Y 580.402,Z 232.058,A -85,B 0,C 180,E1 -1925.777,E2 -1925.777} C_VEL
LIN {X 0,Y 580.259,Z 231.209,A -85,B 0,C 180,E1 -1926.232,E2 -1926.232} C_VEL
LIN {X 0,Y 580.29,Z 231.201,A -85,B 0,C 180,E1 -1929.184,E2 -1929.184} C_VEL
LIN {X 0,Y 580.292,Z 231.204,A -85,B 0,C 180,E1 -1931.768,E2 -1931.768} C_VEL
LIN {X 0,Y 580.259,Z 231.203,A -85,B 0,C 180,E1 -1934.627,E2 -1934.627} C_VEL
LIN {X 0,Y 580.263,Z 231.207,A -85,B 0,C 180,E1 -1937.292,E2 -1937.292} C_VEL
LIN {X 0,Y 580.267,Z 231.202,A -85,B 0,C 180,E1 -1940.065,E2 -1940.065} C_VEL
LIN {X 0,Y 580.276,Z 231.2,A -85,B 0,C 180,E1 -1943.069,E2 -1943.069} C_VEL
LIN {X 0,Y 580.317,Z 231.198,A -85,B 0,C 180,E1 -1946.145,E2 -1946.145} C_VEL
LIN {X 0,Y 580.288,Z 231.2,A -85,B 0,C 180,E1 -1948.615,E2 -1948.615} C_VEL
LIN {X 0,Y 580.287,Z 231.204,A -85,B 0,C 180,E1 -1951.023,E2 -1951.023} C_VEL
LIN {X 0,Y 580.264,Z 231.202,A -85,B 0,C 180,E1 -1953.672,E2 -1953.672} C_VEL
LIN {X 0,Y 580.259,Z 231.204,A -85,B 0,C 180,E1 -1956.441,E2 -1956.441} C_VEL
LIN {X 0,Y 580.276,Z 231.207,A -85,B 0,C 180,E1 -1959.437,E2 -1959.437} C_VEL
LIN {X 0,Y 580.27,Z 231.203,A -85,B 0,C 180,E1 -1961.645,E2 -1961.645} C_VEL
LIN {X 0,Y 580.27,Z 231.202,A -85,B 0,C 180,E1 -1963.825,E2 -1963.825} C_VEL
LIN {X 0,Y 580.314,Z 231.199,A -85,B 0,C 180,E1 -1965.983,E2 -1965.983} C_VEL
LIN {X 0,Y 580.308,Z 231.196,A -85,B 0,C 180,E1 -1968.827,E2 -1968.827} C_VEL
LIN {X 0,Y 580.298,Z 231.202,A -85,B 0,C 180,E1 -1971.643,E2 -1971.643} C_VEL
LIN {X 0,Y 580.276,Z 231.201,A -85,B 0,C 180,E1 -1973.742,E2 -1973.742} C_VEL
LIN {X 0,Y 580.268,Z 231.202,A -85,B 0,C 180,E1 -1975.833,E2 -1975.833} C_VEL
LIN {X 0,Y 580.34,Z 231.195,A -85,B 0,C 180,E1 -1977.918,E2 -1977.918} C_VEL
LIN {X 0,Y 580.345,Z 231.192,A -85,B 0,C 180,E1 -1980.694,E2 -1980.694} C_VEL
LIN {X 0,Y 580.266,Z 231.208,A -85,B 0,C 180,E1 -1983.472,E2 -1983.472} C_VEL
LIN {X 0,Y 580.316,Z 231.197,A -85,B 0,C 180,E1 -1985.56,E2 -1985.56} C_VEL
LIN {X 0,Y 580.308,Z 231.201,A -85,B 0,C 180,E1 -1988.356,E2 -1988.356} C_VEL
LIN {X 0,Y 580.303,Z 231.197,A -85,B 0,C 180,E1 -1991.191,E2 -1991.191} C_VEL
LIN {X 0,Y 580.31,Z 231.2,A -85,B 0,C 180,E1 -1994.017,E2 -1994.017} C_VEL
LIN {X 0,Y 580.292,Z 231.203,A -85,B 0,C 180,E1 -1996.906,E2 -1996.906} C_VEL
LIN {X 0,Y 580.281,Z 231.2,A -85,B 0,C 180,E1 -1999.823,E2 -1999.823} C_VEL
LIN {X 0,Y 580.286,Z 231.199,A -85,B 0,C 180,E1 -2001.313,E2 -2001.313} C_VEL
LIN {X 0,Y 579.586,Z 231.29,A -85,B 0,C 180,E1 -2001.892,E2 -2001.892} C_VEL
LIN {X 0,Y 576.708,Z 231.646,A -85,B 0,C 180,E1 -2002.832,E2 -2002.832} C_VEL
LIN {X 0,Y 574.314,Z 231.945,A -85,B 0,C 180,E1 -2003.588,E2 -2003.588} C_VEL
LIN {X 0,Y 573.316,Z 232.072,A -85,B 0,C 180,E1 -2004.172,E2 -2004.172} C_VEL
LIN {X 0,Y 573.25,Z 232.076,A -85,B 0,C 180,E1 -2004.37,E2 -2004.37} C_VEL
LIN {X 0,Y 573.252,Z 232.078,A -85,B 0,C 180,E1 -2006.976,E2 -2006.976} C_VEL
LIN {X 0,Y 573.219,Z 232.082,A -85,B 0,C 180,E1 -2009.483,E2 -2009.483} C_VEL
LIN {X 0,Y 573.249,Z 232.082,A -85,B 0,C 180,E1 -2012.646,E2 -2012.646} C_VEL
LIN {X 0,Y 573.195,Z 232.082,A -85,B 0,C 180,E1 -2015.189,E2 -2015.189} C_VEL
LIN {X 0,Y 573.233,Z 232.084,A -85,B 0,C 180,E1 -2017.808,E2 -2017.808} C_VEL
LIN {X 0,Y 573.247,Z 232.077,A -85,B 0,C 180,E1 -2020.525,E2 -2020.525} C_VEL
LIN {X 0,Y 573.212,Z 232.082,A -85,B 0,C 180,E1 -2023.362,E2 -2023.362} C_VEL
LIN {X 0,Y 573.197,Z 232.088,A -85,B 0,C 180,E1 -2026.336,E2 -2026.336} C_VEL
LIN {X 0,Y 573.205,Z 232.082,A -85,B 0,C 180,E1 -2028.541,E2 -2028.541} C_VEL
LIN {X 0,Y 573.242,Z 232.082,A -85,B 0,C 180,E1 -2031.298,E2 -2031.298} C_VEL
LIN {X 0,Y 573.193,Z 232.083,A -85,B 0,C 180,E1 -2033.947,E2 -2033.947} C_VEL
LIN {X 0,Y 573.186,Z 232.298,A -85,B 0,C 180,E1 -2034.811,E2 -2034.811} C_VEL
LIN {X 0,Y 573.172,Z 236.464,A -85,B 0,C 180,E1 -2037.35,E2 -2037.35} C_VEL
LIN {X 0,Y 573.126,Z 240.535,A -85,B 0,C 180,E1 -2039.817,E2 -2039.817} C_VEL
LIN {X 0,Y 573.152,Z 244.581,A -85,B 0,C 180,E1 -2042.228,E2 -2042.228} C_VEL
LIN {X 0,Y 573.077,Z 249.984,A -85,B 0,C 180,E1 -2045.357,E2 -2045.357} C_VEL
LIN {X 0,Y 573.043,Z 254.011,A -85,B 0,C 180,E1 -2047.654,E2 -2047.654} C_VEL
LIN {X 0,Y 573.016,Z 258.101,A -85,B 0,C 180,E1 -2049.915,E2 -2049.915} C_VEL
LIN {X 0,Y 572.986,Z 262.248,A -85,B 0,C 180,E1 -2052.143,E2 -2052.143} C_VEL
LIN {X 0,Y 573.002,Z 267.778,A -85,B 0,C 180,E1 -2055.074,E2 -2055.074} C_VEL
LIN {X 0,Y 573.013,Z 272.53,A -85,B 0,C 180,E1 -2057.561,E2 -2057.561} C_VEL
LIN {X 0,Y 573.861,Z 279.429,A -85,B 0,C 180,E1 -2057.737,E2 -2057.737} C_VEL
LIN {X 0,Y 573.734,Z 292.469,A -85,B 0,C 180,E1 -2058.115,E2 -2058.115} C_VEL
LIN {X 0,Y 573.651,Z 304.663,A -85,B 0,C 180,E1 -2058.615,E2 -2058.615} C_VEL
LIN {X 0,Y 573.52,Z 316.044,A -85,B 0,C 180,E1 -2059.23,E2 -2059.23} C_VEL
LIN {X 0,Y 573.389,Z 327.674,A -85,B 0,C 180,E1 -2060.03,E2 -2060.03} C_VEL
LIN {X 0,Y 573.287,Z 337.051,A -85,B 0,C 180,E1 -2060.83,E2 -2060.83} C_VEL
LIN {X 0,Y 573.201,Z 345.611,A -85,B 0,C 180,E1 -2061.717,E2 -2061.717} C_VEL
LIN {X 0,Y 573.138,Z 353.924,A -85,B 0,C 180,E1 -2062.78,E2 -2062.78} C_VEL
LIN {X 0,Y 573.065,Z 360.621,A -85,B 0,C 180,E1 -2063.84,E2 -2063.84} C_VEL
LIN {X 0,Y 572.963,Z 366.763,A -85,B 0,C 180,E1 -2065.074,E2 -2065.074} C_VEL
LIN {X 0,Y 573.014,Z 370.752,A -85,B 0,C 180,E1 -2066.132,E2 -2066.132} C_VEL
LIN {X 0,Y 572.959,Z 373.701,A -85,B 0,C 180,E1 -2067.188,E2 -2067.188} C_VEL
LIN {X 0,Y 572.938,Z 375.128,A -85,B 0,C 180,E1 -2067.891,E2 -2067.891} C_VEL
LIN {X 0,Y 572.941,Z 376.755,A -85,B 0,C 180,E1 -2069.297,E2 -2069.297} C_VEL
LIN {X 0,Y 572.938,Z 376.996,A -85,B 0,C 180,E1 -2070,E2 -2070} C_VEL
LIN {X 0,Y 572.94,Z 376.815,A -85,B 0,C 180,E1 -2070.703,E2 -2070.703} C_VEL
LIN {X 0,Y 572.937,Z 375.27,A -85,B 0,C 180,E1 -2072.109,E2 -2072.109} C_VEL
LIN {X 0,Y 572.96,Z 373.909,A -85,B 0,C 180,E1 -2072.812,E2 -2072.812} C_VEL
LIN {X 0,Y 573.014,Z 371.032,A -85,B 0,C 180,E1 -2073.868,E2 -2073.868} C_VEL
LIN {X 0,Y 572.963,Z 367.131,A -85,B 0,C 180,E1 -2074.926,E2 -2074.926} C_VEL
LIN {X 0,Y 573.075,Z 362.099,A -85,B 0,C 180,E1 -2075.984,E2 -2075.984} C_VEL
LIN {X 0,Y 573.083,Z 355.775,A -85,B 0,C 180,E1 -2077.044,E2 -2077.044} C_VEL
LIN {X 0,Y 573.175,Z 347.854,A -85,B 0,C 180,E1 -2078.106,E2 -2078.106} C_VEL
LIN {X 0,Y 573.287,Z 338.004,A -85,B 0,C 180,E1 -2079.17,E2 -2079.17} C_VEL
LIN {X 0,Y 573.405,Z 327.684,A -85,B 0,C 180,E1 -2080.059,E2 -2080.059} C_VEL
LIN {X 0,Y 573.49,Z 316.09,A -85,B 0,C 180,E1 -2080.858,E2 -2080.858} C_VEL
LIN {X 0,Y 573.658,Z 305.197,A -85,B 0,C 180,E1 -2081.449,E2 -2081.449} C_VEL
LIN {X 0,Y 573.749,Z 292.606,A -85,B 0,C 180,E1 -2081.97,E2 -2081.97} C_VEL
LIN {X 0,Y 573.858,Z 279.437,A -85,B 0,C 180,E1 -2082.353,E2 -2082.353} C_VEL
LIN {X 0,Y 573.207,Z 274.082,A -85,B 0,C 180,E1 -2082.48,E2 -2082.48} C_VEL
LIN {X 0,Y 572.986,Z 272.53,A -85,B 0,C 180,E1 -2082.53,E2 -2082.53} C_VEL
LIN {X 0,Y 573.003,Z 267.949,A -85,B 0,C 180,E1 -2084.926,E2 -2084.926} C_VEL
LIN {X 0,Y 572.987,Z 262.416,A -85,B 0,C 180,E1 -2087.857,E2 -2087.857} C_VEL
LIN {X 0,Y 573.016,Z 258.267,A -85,B 0,C 180,E1 -2090.085,E2 -2090.085} C_VEL
LIN {X 0,Y 573.091,Z 252.818,A -85,B 0,C 180,E1 -2093.11,E2 -2093.11} C_VEL
LIN {X 0,Y 573.085,Z 248.801,A -85,B 0,C 180,E1 -2095.418,E2 -2095.418} C_VEL
LIN {X 0,Y 573.153,Z 243.386,A -85,B 0,C 180,E1 -2098.569,E2 -2098.569} C_VEL
LIN {X 0,Y 573.138,Z 239.331,A -85,B 0,C 180,E1 -2100.999,E2 -2100.999} C_VEL
LIN {X 0,Y 573.175,Z 235.195,A -85,B 0,C 180,E1 -2103.51,E2 -2103.51} C_VEL
LIN {X 0,Y 573.185,Z 232.445,A -85,B 0,C 180,E1 -2105.19,E2 -2105.19} C_VEL
LIN {X 0,Y 573.195,Z 232.083,A -85,B 0,C 180,E1 -2106.053,E2 -2106.053} C_VEL
LIN {X 0,Y 573.244,Z 232.083,A -85,B 0,C 180,E1 -2108.702,E2 -2108.702} C_VEL
LIN {X 0,Y 573.215,Z 232.081,A -85,B 0,C 180,E1 -2111.591,E2 -2111.591} C_VEL
LIN {X 0,Y 573.197,Z 232.083,A -85,B 0,C 180,E1 -2114.672,E2 -2114.672} C_VEL
LIN {X 0,Y 573.241,Z 232.08,A -85,B 0,C 180,E1 -2117.599,E2 -2117.599} C_VEL
LIN {X 0,Y 573.244,Z 232.083,A -85,B 0,C 180,E1 -2120.569,E2 -2120.569} C_VEL
LIN {X 0,Y 573.256,Z 232.075,A -85,B 0,C 180,E1 -2123.078,E2 -2123.078} C_VEL
LIN {X 0,Y 573.254,Z 232.08,A -85,B 0,C 180,E1 -2125.67,E2 -2125.67} C_VEL
LIN {X 0,Y 573.237,Z 232.078,A -85,B 0,C 180,E1 -2128.184,E2 -2128.184} C_VEL
LIN {X 0,Y 573.239,Z 232.081,A -85,B 0,C 180,E1 -2130.633,E2 -2130.633} C_VEL
LIN {X 0,Y 573.253,Z 232.078,A -85,B 0,C 180,E1 -2133.024,E2 -2133.024} C_VEL
LIN {X 0,Y 573.279,Z 232.072,A -85,B 0,C 180,E1 -2135.366,E2 -2135.366} C_VEL
LIN {X 0,Y 573.232,Z 232.078,A -85,B 0,C 180,E1 -2138.419,E2 -2138.419} C_VEL
LIN {X 0,Y 573.273,Z 232.074,A -85,B 0,C 180,E1 -2140.731,E2 -2140.731} C_VEL
LIN {X 0,Y 573.223,Z 232.08,A -85,B 0,C 180,E1 -2143.621,E2 -2143.621} C_VEL
LIN {X 0,Y 573.254,Z 232.077,A -85,B 0,C 180,E1 -2145.806,E2 -2145.806} C_VEL
LIN {X 0,Y 573.267,Z 232.074,A -85,B 0,C 180,E1 -2148.745,E2 -2148.745} C_VEL
LIN {X 0,Y 573.252,Z 232.082,A -85,B 0,C 180,E1 -2151.54,E2 -2151.54} C_VEL
LIN {X 0,Y 573.213,Z 232.081,A -85,B 0,C 180,E1 -2153.665,E2 -2153.665} C_VEL
LIN {X 0,Y 573.191,Z 232.083,A -85,B 0,C 180,E1 -2155.781,E2 -2155.781} C_VEL
LIN {X 0,Y 573.291,Z 232.072,A -85,B 0,C 180,E1 -2157.892,E2 -2157.892} C_VEL
LIN {X 0,Y 573.331,Z 232.066,A -85,B 0,C 180,E1 -2160.702,E2 -2160.702} C_VEL
LIN {X 0,Y 573.308,Z 232.069,A -85,B 0,C 180,E1 -2162.811,E2 -2162.811} C_VEL
LIN {X 0,Y 573.289,Z 232.073,A -85,B 0,C 180,E1 -2165.628,E2 -2165.628} C_VEL
LIN {X 0,Y 573.242,Z 232.076,A -85,B 0,C 180,E1 -2167.751,E2 -2167.751} C_VEL
LIN {X 0,Y 573.225,Z 232.082,A -85,B 0,C 180,E1 -2170.597,E2 -2170.597} C_VEL
LIN {X 0,Y 573.219,Z 232.083,A -85,B 0,C 180,E1 -2173.471,E2 -2173.471} C_VEL
LIN {X 0,Y 573.228,Z 232.084,A -85,B 0,C 180,E1 -2175.648,E2 -2175.648} C_VEL
LIN {X 0,Y 573.247,Z 232.077,A -85,B 0,C 180,E1 -2177.848,E2 -2177.848} C_VEL
LIN {X 0,Y 573.246,Z 232.078,A -85,B 0,C 180,E1 -2180.077,E2 -2180.077} C_VEL
LIN {X 0,Y 573.234,Z 232.084,A -85,B 0,C 180,E1 -2182.338,E2 -2182.338} C_VEL
LIN {X 0,Y 573.226,Z 232.081,A -85,B 0,C 180,E1 -2185.411,E2 -2185.411} C_VEL
LIN {X 0,Y 573.224,Z 232.08,A -85,B 0,C 180,E1 -2188.565,E2 -2188.565} C_VEL
LIN {X 0,Y 573.227,Z 232.085,A -85,B 0,C 180,E1 -2190.993,E2 -2190.993} C_VEL
LIN {X 0,Y 573.266,Z 232.074,A -85,B 0,C 180,E1 -2193.524,E2 -2193.524} C_VEL
LIN {X 0,Y 573.195,Z 232.089,A -85,B 0,C 180,E1 -2196.053,E2 -2196.053} C_VEL
LIN {X 0,Y 573.229,Z 232.078,A -85,B 0,C 180,E1 -2198.703,E2 -2198.703} C_VEL
LIN {X 0,Y 573.212,Z 232.082,A -85,B 0,C 180,E1 -2201.59,E2 -2201.59} C_VEL
LIN {X 0,Y 573.225,Z 232.083,A -85,B 0,C 180,E1 -2204.335,E2 -2204.335} C_VEL
LIN {X 0,Y 573.243,Z 232.077,A -85,B 0,C 180,E1 -2207.358,E2 -2207.358} C_VEL
LIN {X 0,Y 573.238,Z 232.079,A -85,B 0,C 180,E1 -2210.392,E2 -2210.392} C_VEL
LIN {X 0,Y 573.233,Z 232.085,A -85,B 0,C 180,E1 -2213.076,E2 -2213.076} C_VEL
LIN {X 0,Y 573.243,Z 232.092,A -85,B 0,C 180,E1 -2213.733,E2 -2213.733} C_VEL
LIN {X 0,Y 573.52,Z 235.738,A -85,B 0,C 180,E1 -2215.188,E2 -2215.188} C_VEL
LIN {X 0,Y 573.479,Z 242.425,A -85,B 0,C 180,E1 -2217.736,E2 -2217.736} C_VEL
LIN {X 0,Y 573.361,Z 250.448,A -85,B 0,C 180,E1 -2220.639,E2 -2220.639} C_VEL
LIN {X 0,Y 573.274,Z 258.553,A -85,B 0,C 180,E1 -2223.501,E2 -2223.501} C_VEL
LIN {X 0,Y 573.262,Z 266.239,A -85,B 0,C 180,E1 -2226.136,E2 -2226.136} C_VEL
LIN {X 0,Y 573.236,Z 273.881,A -85,B 0,C 180,E1 -2228.714,E2 -2228.714} C_VEL
LIN {X 0,Y 573.159,Z 281.917,A -85,B 0,C 180,E1 -2231.409,E2 -2231.409} C_VEL
LIN {X 0,Y 573.107,Z 290.822,A -85,B 0,C 180,E1 -2234.348,E2 -2234.348} C_VEL
LIN {X 0,Y 573.065,Z 299.726,A -85,B 0,C 180,E1 -2237.247,E2 -2237.247} C_VEL
LIN {X 0,Y 573.045,Z 300.491,A -85,B 0,C 180,E1 -2237.494,E2 -2237.494} C_VEL
LIN {X 0,Y 573.875,Z 306.363,A -85,B 0,C 180,E1 -2237.625,E2 -2237.625} C_VEL
LIN {X 0,Y 573.771,Z 318.495,A -85,B 0,C 180,E1 -2237.936,E2 -2237.936} C_VEL
LIN {X 0,Y 573.65,Z 330.314,A -85,B 0,C 180,E1 -2238.373,E2 -2238.373} C_VEL
LIN {X 0,Y 573.511,Z 342.645,A -85,B 0,C 180,E1 -2238.986,E2 -2238.986} C_VEL
LIN {X 0,Y 573.442,Z 353.48,A -85,B 0,C 180,E1 -2239.674,E2 -2239.674} C_VEL
LIN {X 0,Y 573.308,Z 363.646,A -85,B 0,C 180,E1 -2240.474,E2 -2240.474} C_VEL
LIN {X 0,Y 573.215,Z 372.786,A -85,B 0,C 180,E1 -2241.362,E2 -2241.362} C_VEL
LIN {X 0,Y 573.142,Z 381.689,A -85,B 0,C 180,E1 -2242.425,E2 -2242.425} C_VEL
LIN {X 0,Y 573.051,Z 388.404,A -85,B 0,C 180,E1 -2243.415,E2 -2243.415} C_VEL
LIN {X 0,Y 573.07,Z 393.679,A -85,B 0,C 180,E1 -2244.37,E2 -2244.37} C_VEL
LIN {X 0,Y 573.028,Z 398.372,A -85,B 0,C 180,E1 -2245.427,E2 -2245.427} C_VEL
LIN {X 0,Y 573.022,Z 401.957,A -85,B 0,C 180,E1 -2246.484,E2 -2246.484} C_VEL
LIN {X 0,Y 572.959,Z 403.808,A -85,B 0,C 180,E1 -2247.188,E2 -2247.188} C_VEL
LIN {X 0,Y 572.94,Z 405.198,A -85,B 0,C 180,E1 -2247.891,E2 -2247.891} C_VEL
LIN {X 0,Y 572.94,Z 406.785,A -85,B 0,C 180,E1 -2249.297,E2 -2249.297} C_VEL
LIN {X 0,Y 572.938,Z 407,A -85,B 0,C 180,E1 -2250,E2 -2250} C_VEL
LIN {X 0,Y 572.946,Z 406.186,A -85,B 0,C 180,E1 -2251.406,E2 -2251.406} C_VEL
LIN {X 0,Y 572.94,Z 405.2,A -85,B 0,C 180,E1 -2252.109,E2 -2252.109} C_VEL
LIN {X 0,Y 572.959,Z 403.81,A -85,B 0,C 180,E1 -2252.812,E2 -2252.812} C_VEL
LIN {X 0,Y 573.014,Z 400.896,A -85,B 0,C 180,E1 -2253.868,E2 -2253.868} C_VEL
LIN {X 0,Y 572.963,Z 396.949,A -85,B 0,C 180,E1 -2254.926,E2 -2254.926} C_VEL
LIN {X 0,Y 573.065,Z 390.877,A -85,B 0,C 180,E1 -2256.16,E2 -2256.16} C_VEL
LIN {X 0,Y 573.119,Z 384.238,A -85,B 0,C 180,E1 -2257.221,E2 -2257.221} C_VEL
LIN {X 0,Y 573.201,Z 375.991,A -85,B 0,C 180,E1 -2258.283,E2 -2258.283} C_VEL
LIN {X 0,Y 573.287,Z 367.539,A -85,B 0,C 180,E1 -2259.17,E2 -2259.17} C_VEL
LIN {X 0,Y 573.421,Z 357.099,A -85,B 0,C 180,E1 -2260.058,E2 -2260.058} C_VEL
LIN {X 0,Y 573.519,Z 345.535,A -85,B 0,C 180,E1 -2260.847,E2 -2260.847} C_VEL
LIN {X 0,Y 573.609,Z 333.884,A -85,B 0,C 180,E1 -2261.466,E2 -2261.466} C_VEL
LIN {X 0,Y 573.763,Z 321.172,A -85,B 0,C 180,E1 -2261.974,E2 -2261.974} C_VEL
LIN {X 0,Y 573.854,Z 308.52,A -85,B 0,C 180,E1 -2262.331,E2 -2262.331} C_VEL
LIN {X 0,Y 573.68,Z 304.532,A -85,B 0,C 180,E1 -2262.416,E2 -2262.416} C_VEL
LIN {X 0,Y 573.045,Z 300.492,A -85,B 0,C 180,E1 -2262.506,E2 -2262.506} C_VEL
LIN {X 0,Y 573.085,Z 291.935,A -85,B 0,C 180,E1 -2265.288,E2 -2265.288} C_VEL
LIN {X 0,Y 573.146,Z 284.144,A -85,B 0,C 180,E1 -2267.852,E2 -2267.852} C_VEL
LIN {X 0,Y 573.196,Z 276.352,A -85,B 0,C 180,E1 -2270.453,E2 -2270.453} C_VEL
LIN {X 0,Y 573.216,Z 268.388,A -85,B 0,C 180,E1 -2273.139,E2 -2273.139} C_VEL
LIN {X 0,Y 573.28,Z 260.573,A -85,B 0,C 180,E1 -2275.798,E2 -2275.798} C_VEL
LIN {X 0,Y 573.33,Z 252.699,A -85,B 0,C 180,E1 -2278.559,E2 -2278.559} C_VEL
LIN {X 0,Y 573.399,Z 244.809,A -85,B 0,C 180,E1 -2281.393,E2 -2281.393} C_VEL
LIN {X 0,Y 573.474,Z 239.017,A -85,B 0,C 180,E1 -2283.555,E2 -2283.555} C_VEL
LIN {X 0,Y 573.494,Z 233.789,A -85,B 0,C 180,E1 -2285.576,E2 -2285.576} C_VEL
LIN {X 0,Y 573.226,Z 232.085,A -85,B 0,C 180,E1 -2286.323,E2 -2286.323} C_VEL
LIN {X 0,Y 573.237,Z 232.084,A -85,B 0,C 180,E1 -2288.702,E2 -2288.702} C_VEL
